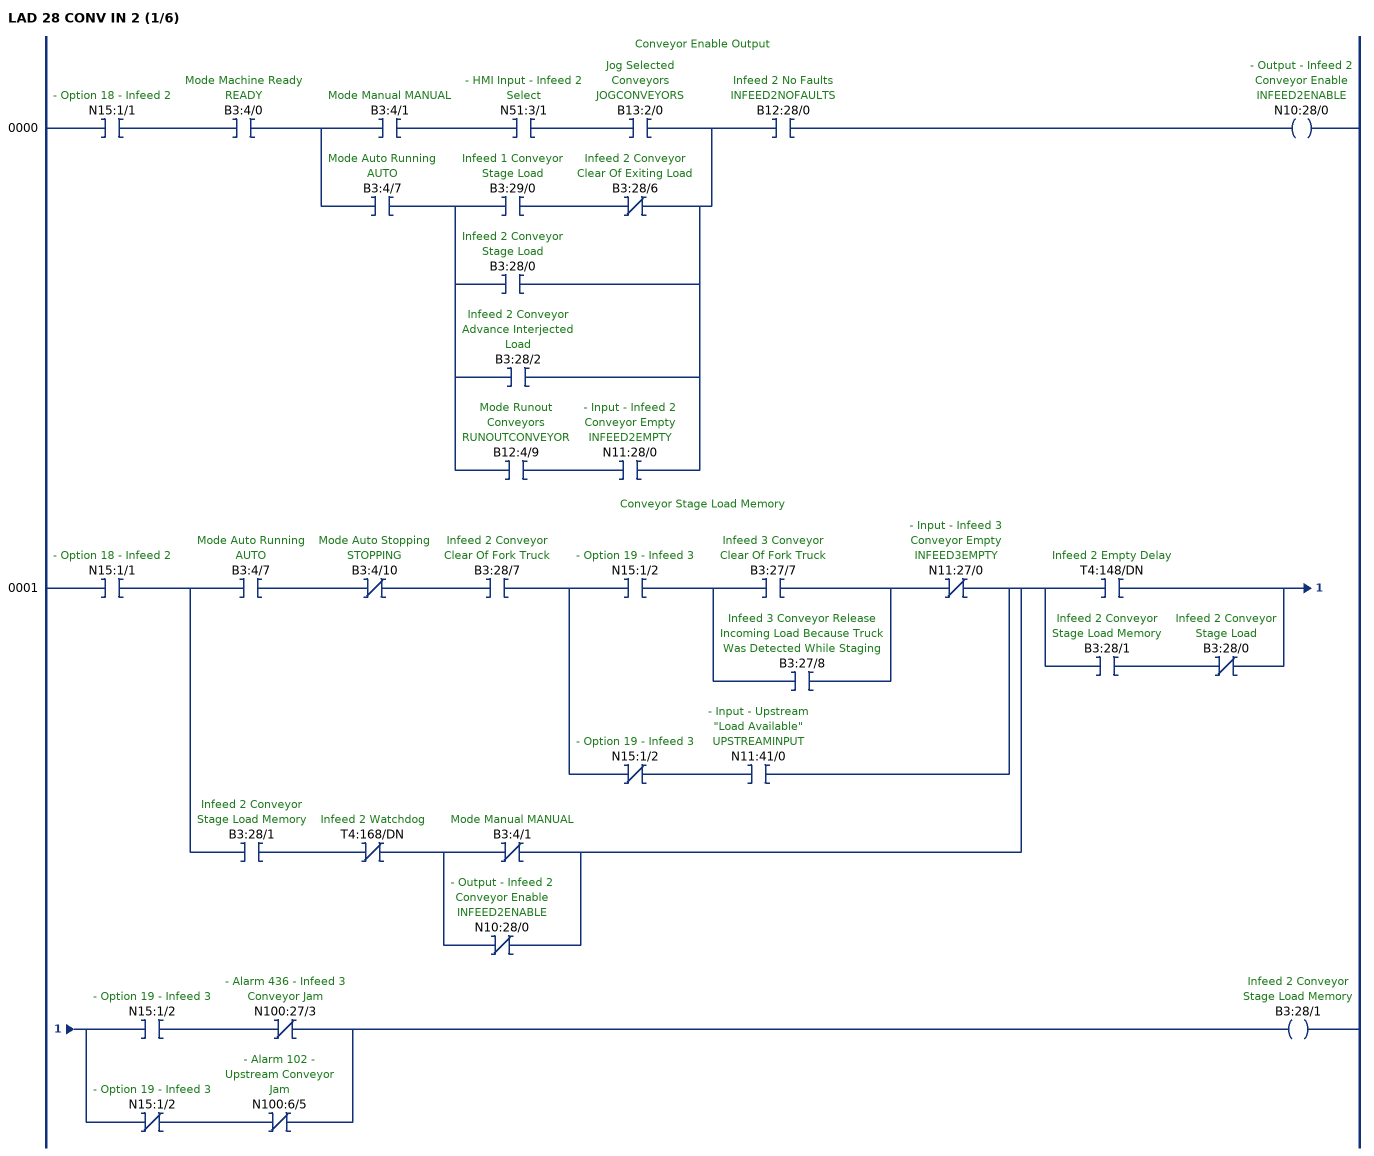
% Rung: 0 %
% Conveyor Enable Output %
SOR XIC N15:1/1 XIC B3:4/0 BST XIC B3:4/1 XIC N51:3/1 XIC B13:2/0 NXB XIC B3:4/7 BST XIC B3:29/0 XIO B3:28/6 NXB XIC B3:28/0 NXB XIC B3:28/2 NXB XIC B12:4/9 XIC N11:28/0 BND BND XIC B12:28/0 OTE N10:28/0 EOR
%   N15:1/1  "- Option 18 - Infeed 2" %
%   B3:4/0  READY  "Mode Machine Ready" %
%   B3:4/1  MANUAL  "Mode Manual" %
%   N51:3/1  "- HMI Input - Infeed 2 Select" %
%   B13:2/0  JOGCONVEYORS  "Jog Selected Conveyors" %
%   B3:4/7  AUTO  "Mode Auto Running" %
%   B3:29/0  "Infeed 1 Conveyor Stage Load" %
%   B3:28/6  "Infeed 2 Conveyor Clear Of Exiting Load" %
%   B3:28/0  "Infeed 2 Conveyor Stage Load" %
%   B3:28/2  "Infeed 2 Conveyor Advance Interjected Load" %
%   B12:4/9  RUNOUTCONVEYOR  "Mode Runout Conveyors" %
%   N11:28/0  INFEED2EMPTY  "- Input - Infeed 2 Conveyor Empty" %
%   B12:28/0  INFEED2NOFAULTS  "Infeed 2 No Faults" %
%   N10:28/0  INFEED2ENABLE  "- Output - Infeed 2 Conveyor Enable" %
% Rung: 1 %
% Conveyor Stage Load Memory %
SOR XIC N15:1/1 BST XIC B3:4/7 XIO B3:4/10 XIC B3:28/7 BST XIC N15:1/2 BST XIC B3:27/7 NXB XIC B3:27/8 BND XIO N11:27/0 NXB XIO N15:1/2 XIC N11:41/0 BND NXB XIC B3:28/1 XIO T4:168/DN BST XIO B3:4/1 NXB XIO N10:28/0 BND BND BST XIC T4:148/DN NXB XIC B3:28/1 XIO B3:28/0 BND BST XIC N15:1/2 XIO N100:27/3 NXB XIO N15:1/2 XIO N100:6/5 BND OTE B3:28/1 EOR
%   N15:1/1  "- Option 18 - Infeed 2" %
%   B3:4/7  AUTO  "Mode Auto Running" %
%   B3:4/10  STOPPING  "Mode Auto Stopping" %
%   B3:28/7  "Infeed 2 Conveyor Clear Of Fork Truck" %
%   N15:1/2  "- Option 19 - Infeed 3" %
%   B3:27/7  "Infeed 3 Conveyor Clear Of Fork Truck" %
%   B3:27/8  "Infeed 3 Conveyor Release Incoming Load Because Truck Was Detected While Staging" %
%   N11:27/0  INFEED3EMPTY  "- Input - Infeed 3 Conveyor Empty" %
%   N11:41/0  UPSTREAMINPUT  "- Input - Upstream "Load Available"" %
%   B3:28/1  "Infeed 2 Conveyor Stage Load Memory" %
%   T4:168  "Infeed 2 Watchdog" %
%   B3:4/1  MANUAL  "Mode Manual" %
%   N10:28/0  INFEED2ENABLE  "- Output - Infeed 2 Conveyor Enable" %
%   T4:148  "Infeed 2 Empty Delay" %
%   B3:28/0  "Infeed 2 Conveyor Stage Load" %
%   N100:27/3  "- Alarm 436 - Infeed 3 Conveyor Jam" %
%   N100:6/5  "- Alarm 102 - Upstream Conveyor Jam" %

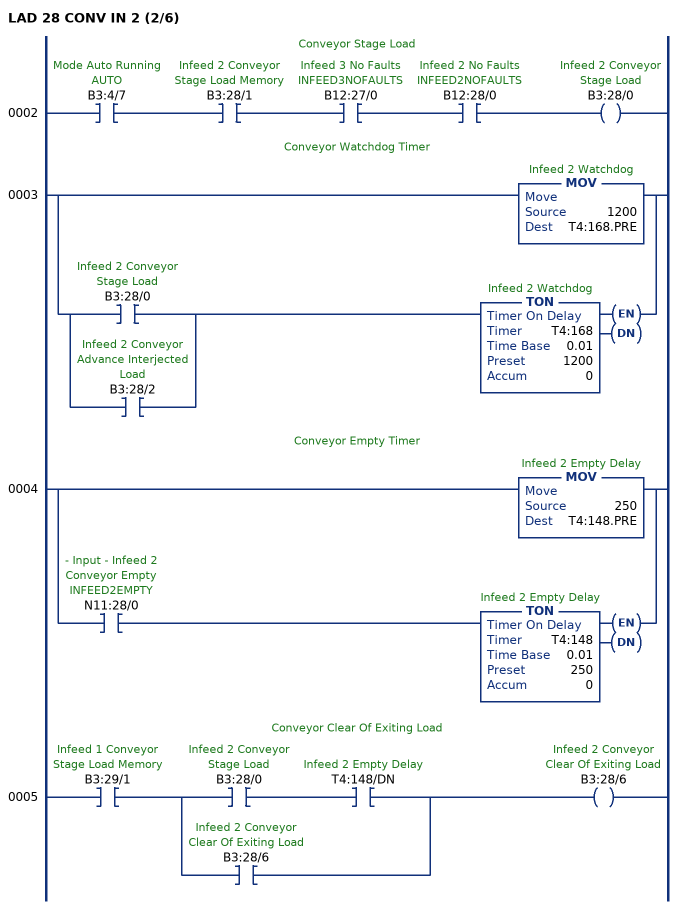
% Rung: 2 %
% Conveyor Stage Load %
SOR XIC B3:4/7 XIC B3:28/1 XIC B12:27/0 XIC B12:28/0 OTE B3:28/0 EOR
%   B3:4/7  AUTO  "Mode Auto Running" %
%   B3:28/1  "Infeed 2 Conveyor Stage Load Memory" %
%   B12:27/0  INFEED3NOFAULTS  "Infeed 3 No Faults" %
%   B12:28/0  INFEED2NOFAULTS  "Infeed 2 No Faults" %
%   B3:28/0  "Infeed 2 Conveyor Stage Load" %
% Rung: 3 %
% Conveyor Watchdog Timer %
SOR BST MOV 1200 T4:168.PRE NXB BST XIC B3:28/0 NXB XIC B3:28/2 BND TON T4:168 0.01 1200 0 BND EOR
%   T4:168  "Infeed 2 Watchdog" %
%   B3:28/0  "Infeed 2 Conveyor Stage Load" %
%   B3:28/2  "Infeed 2 Conveyor Advance Interjected Load" %
% Rung: 4 %
% Conveyor Empty Timer %
SOR BST MOV 250 T4:148.PRE NXB XIC N11:28/0 TON T4:148 0.01 250 0 BND EOR
%   T4:148  "Infeed 2 Empty Delay" %
%   N11:28/0  INFEED2EMPTY  "- Input - Infeed 2 Conveyor Empty" %
% Rung: 5 %
% Conveyor Clear Of Exiting Load %
SOR XIC B3:29/1 BST XIC B3:28/0 XIC T4:148/DN NXB XIC B3:28/6 BND OTE B3:28/6 EOR
%   B3:29/1  "Infeed 1 Conveyor Stage Load Memory" %
%   B3:28/0  "Infeed 2 Conveyor Stage Load" %
%   T4:148  "Infeed 2 Empty Delay" %
%   B3:28/6  "Infeed 2 Conveyor Clear Of Exiting Load" %

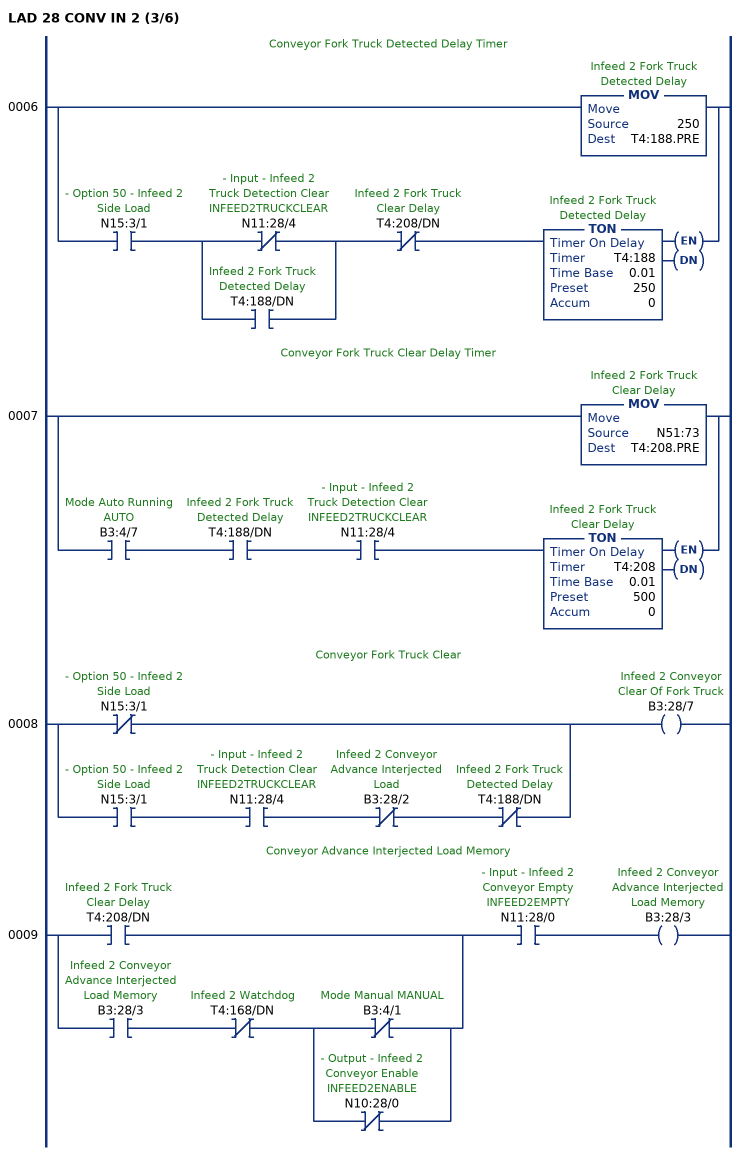
% Rung: 6 %
% Conveyor Fork Truck Detected Delay Timer %
SOR BST MOV 250 T4:188.PRE NXB XIC N15:3/1 BST XIO N11:28/4 NXB XIC T4:188/DN BND XIO T4:208/DN TON T4:188 0.01 250 0 BND EOR
%   T4:188  "Infeed 2 Fork Truck Detected Delay" %
%   N15:3/1  "- Option 50 - Infeed 2 Side Load" %
%   N11:28/4  INFEED2TRUCKCLEAR  "- Input - Infeed 2 Truck Detection Clear" %
%   T4:208  "Infeed 2 Fork Truck Clear Delay" %
% Rung: 7 %
% Conveyor Fork Truck Clear Delay Timer %
SOR BST MOV N51:73 T4:208.PRE NXB XIC B3:4/7 XIC T4:188/DN XIC N11:28/4 TON T4:208 0.01 500 0 BND EOR
%   N51:73  "- HMI Input - Preset Truck Clear" %
%   T4:208  "Infeed 2 Fork Truck Clear Delay" %
%   B3:4/7  AUTO  "Mode Auto Running" %
%   T4:188  "Infeed 2 Fork Truck Detected Delay" %
%   N11:28/4  INFEED2TRUCKCLEAR  "- Input - Infeed 2 Truck Detection Clear" %
% Rung: 8 %
% Conveyor Fork Truck Clear %
SOR BST XIO N15:3/1 NXB XIC N15:3/1 XIC N11:28/4 XIO B3:28/2 XIO T4:188/DN BND OTE B3:28/7 EOR
%   N15:3/1  "- Option 50 - Infeed 2 Side Load" %
%   N11:28/4  INFEED2TRUCKCLEAR  "- Input - Infeed 2 Truck Detection Clear" %
%   B3:28/2  "Infeed 2 Conveyor Advance Interjected Load" %
%   T4:188  "Infeed 2 Fork Truck Detected Delay" %
%   B3:28/7  "Infeed 2 Conveyor Clear Of Fork Truck" %
% Rung: 9 %
% Conveyor Advance Interjected Load Memory %
SOR BST XIC T4:208/DN NXB XIC B3:28/3 XIO T4:168/DN BST XIO B3:4/1 NXB XIO N10:28/0 BND BND XIC N11:28/0 OTE B3:28/3 EOR
%   T4:208  "Infeed 2 Fork Truck Clear Delay" %
%   B3:28/3  "Infeed 2 Conveyor Advance Interjected Load Memory" %
%   T4:168  "Infeed 2 Watchdog" %
%   B3:4/1  MANUAL  "Mode Manual" %
%   N10:28/0  INFEED2ENABLE  "- Output - Infeed 2 Conveyor Enable" %
%   N11:28/0  INFEED2EMPTY  "- Input - Infeed 2 Conveyor Empty" %

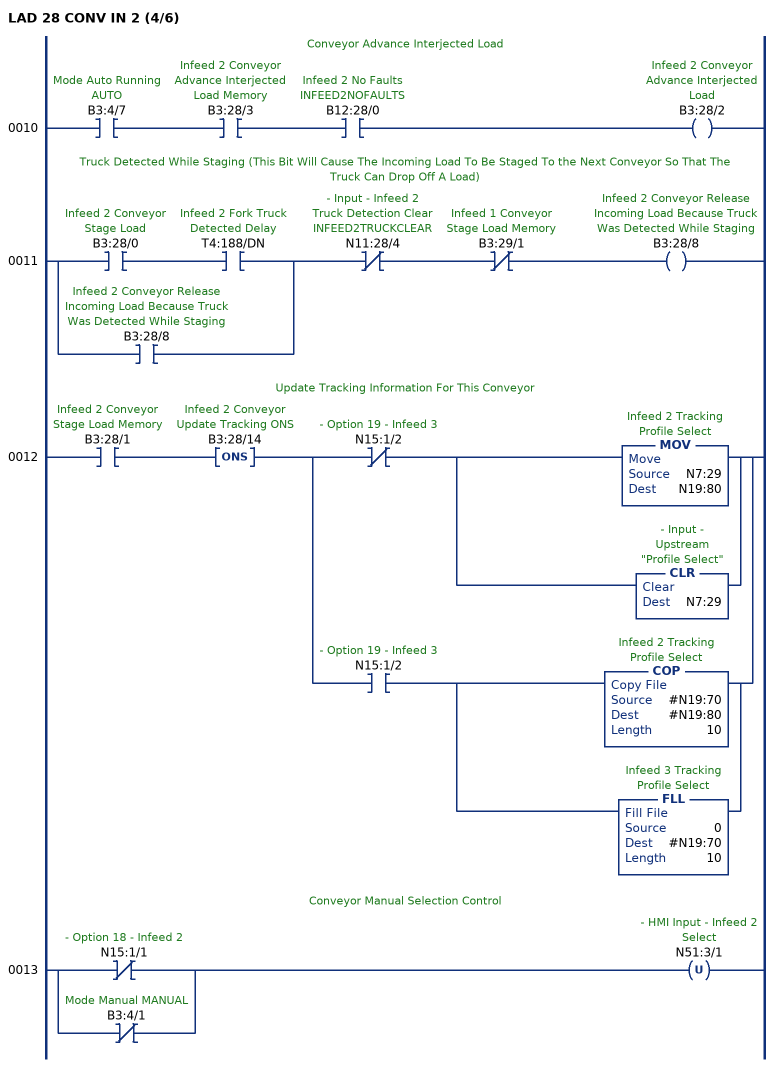
% Rung: 10 %
% Conveyor Advance Interjected Load %
SOR XIC B3:4/7 XIC B3:28/3 XIC B12:28/0 OTE B3:28/2 EOR
%   B3:4/7  AUTO  "Mode Auto Running" %
%   B3:28/3  "Infeed 2 Conveyor Advance Interjected Load Memory" %
%   B12:28/0  INFEED2NOFAULTS  "Infeed 2 No Faults" %
%   B3:28/2  "Infeed 2 Conveyor Advance Interjected Load" %
% Rung: 11 %
% Truck Detected While Staging (This Bit Will Cause The Incoming Load To Be Staged To the Next Conveyor So That The Truck Can Drop Off A Load) %
SOR BST XIC B3:28/0 XIC T4:188/DN NXB XIC B3:28/8 BND XIO N11:28/4 XIO B3:29/1 OTE B3:28/8 EOR
%   B3:28/0  "Infeed 2 Conveyor Stage Load" %
%   T4:188  "Infeed 2 Fork Truck Detected Delay" %
%   B3:28/8  "Infeed 2 Conveyor Release Incoming Load Because Truck Was Detected While Staging" %
%   N11:28/4  INFEED2TRUCKCLEAR  "- Input - Infeed 2 Truck Detection Clear" %
%   B3:29/1  "Infeed 1 Conveyor Stage Load Memory" %
% Rung: 12 %
% Update Tracking Information For This Conveyor %
SOR XIC B3:28/1 ONS B3:28/14 BST XIO N15:1/2 BST MOV N7:29 N19:80 NXB CLR N7:29 BND NXB XIC N15:1/2 BST COP #N19:70 #N19:80 10 NXB FLL 0 #N19:70 10 BND BND EOR
%   B3:28/1  "Infeed 2 Conveyor Stage Load Memory" %
%   B3:28/14  "Infeed 2 Conveyor Update Tracking ONS" %
%   N15:1/2  "- Option 19 - Infeed 3" %
%   N7:29  "- Input - Upstream "Profile Select"" %
%   N19:80  "Infeed 2 Tracking Profile Select" %
%   N19:70  "Infeed 3 Tracking Profile Select" %
% Rung: 13 %
% Conveyor Manual Selection Control %
SOR BST XIO N15:1/1 NXB XIO B3:4/1 BND OTU N51:3/1 EOR
%   N15:1/1  "- Option 18 - Infeed 2" %
%   B3:4/1  MANUAL  "Mode Manual" %
%   N51:3/1  "- HMI Input - Infeed 2 Select" %

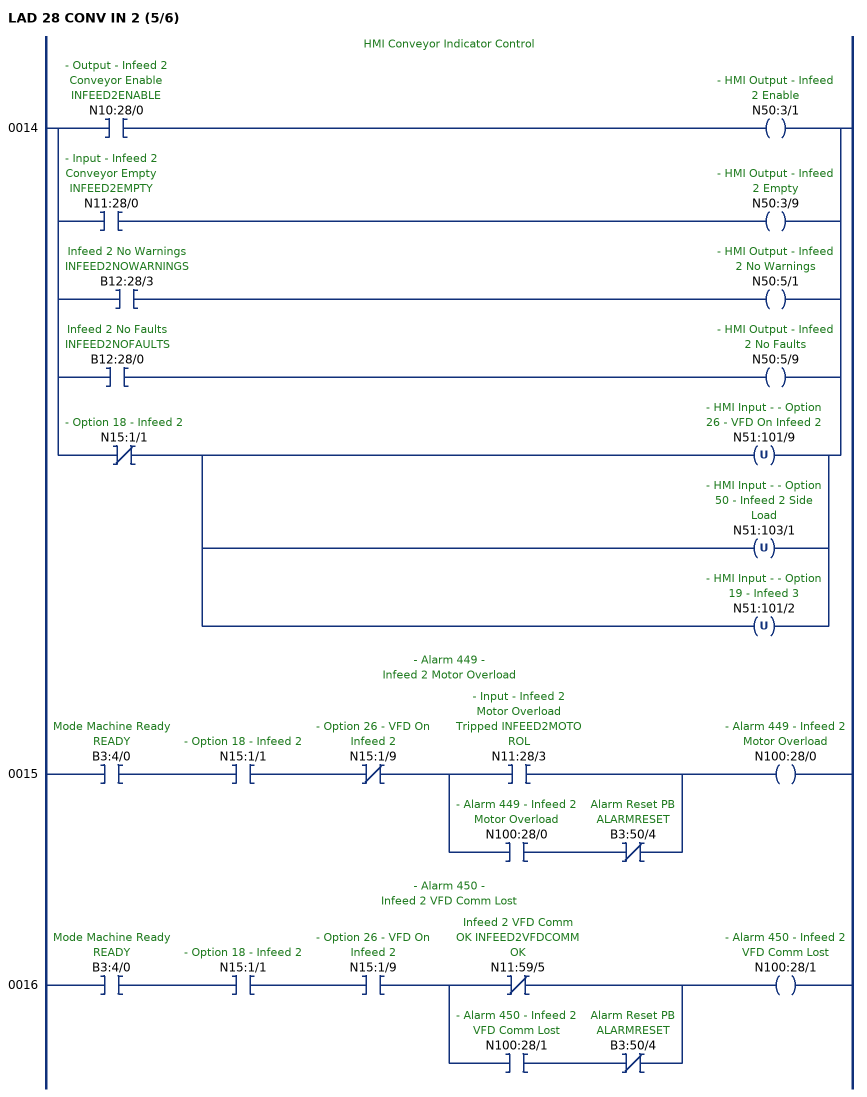
% Rung: 14 %
% HMI Conveyor Indicator Control %
SOR BST XIC N10:28/0 OTE N50:3/1 NXB XIC N11:28/0 OTE N50:3/9 NXB XIC B12:28/3 OTE N50:5/1 NXB XIC B12:28/0 OTE N50:5/9 NXB XIO N15:1/1 BST OTU N51:101/9 NXB OTU N51:103/1 NXB OTU N51:101/2 BND BND EOR
%   N10:28/0  INFEED2ENABLE  "- Output - Infeed 2 Conveyor Enable" %
%   N50:3/1  "- HMI Output - Infeed 2 Enable" %
%   N11:28/0  INFEED2EMPTY  "- Input - Infeed 2 Conveyor Empty" %
%   N50:3/9  "- HMI Output - Infeed 2 Empty" %
%   B12:28/3  INFEED2NOWARNINGS  "Infeed 2 No Warnings" %
%   N50:5/1  "- HMI Output - Infeed 2 No Warnings" %
%   B12:28/0  INFEED2NOFAULTS  "Infeed 2 No Faults" %
%   N50:5/9  "- HMI Output - Infeed 2 No Faults" %
%   N15:1/1  "- Option 18 - Infeed 2" %
%   N51:101/9  "- HMI Input - - Option 26 - VFD On Infeed 2" %
%   N51:103/1  "- HMI Input - - Option 50 - Infeed 2 Side Load" %
%   N51:101/2  "- HMI Input - - Option 19 - Infeed 3" %
% Rung: 15 %
% - Alarm 449 -
% 
% Infeed 2 Motor Overload %
SOR XIC B3:4/0 XIC N15:1/1 XIO N15:1/9 BST XIC N11:28/3 NXB XIC N100:28/0 XIO B3:50/4 BND OTE N100:28/0 EOR
%   B3:4/0  READY  "Mode Machine Ready" %
%   N15:1/1  "- Option 18 - Infeed 2" %
%   N15:1/9  "- Option 26 - VFD On Infeed 2" %
%   N11:28/3  INFEED2MOTOROL  "- Input - Infeed 2 Motor Overload Tripped" %
%   N100:28/0  "- Alarm 449 - Infeed 2 Motor Overload" %
%   B3:50/4  ALARMRESET  "Alarm Reset PB" %
% Rung: 16 %
% - Alarm 450 -
% 
% Infeed 2 VFD Comm Lost %
SOR XIC B3:4/0 XIC N15:1/1 XIC N15:1/9 BST XIO N11:59/5 NXB XIC N100:28/1 XIO B3:50/4 BND OTE N100:28/1 EOR
%   B3:4/0  READY  "Mode Machine Ready" %
%   N15:1/1  "- Option 18 - Infeed 2" %
%   N15:1/9  "- Option 26 - VFD On Infeed 2" %
%   N11:59/5  INFEED2VFDCOMMOK  "Infeed 2 VFD Comm OK" %
%   N100:28/1  "- Alarm 450 - Infeed 2 VFD Comm Lost" %
%   B3:50/4  ALARMRESET  "Alarm Reset PB" %

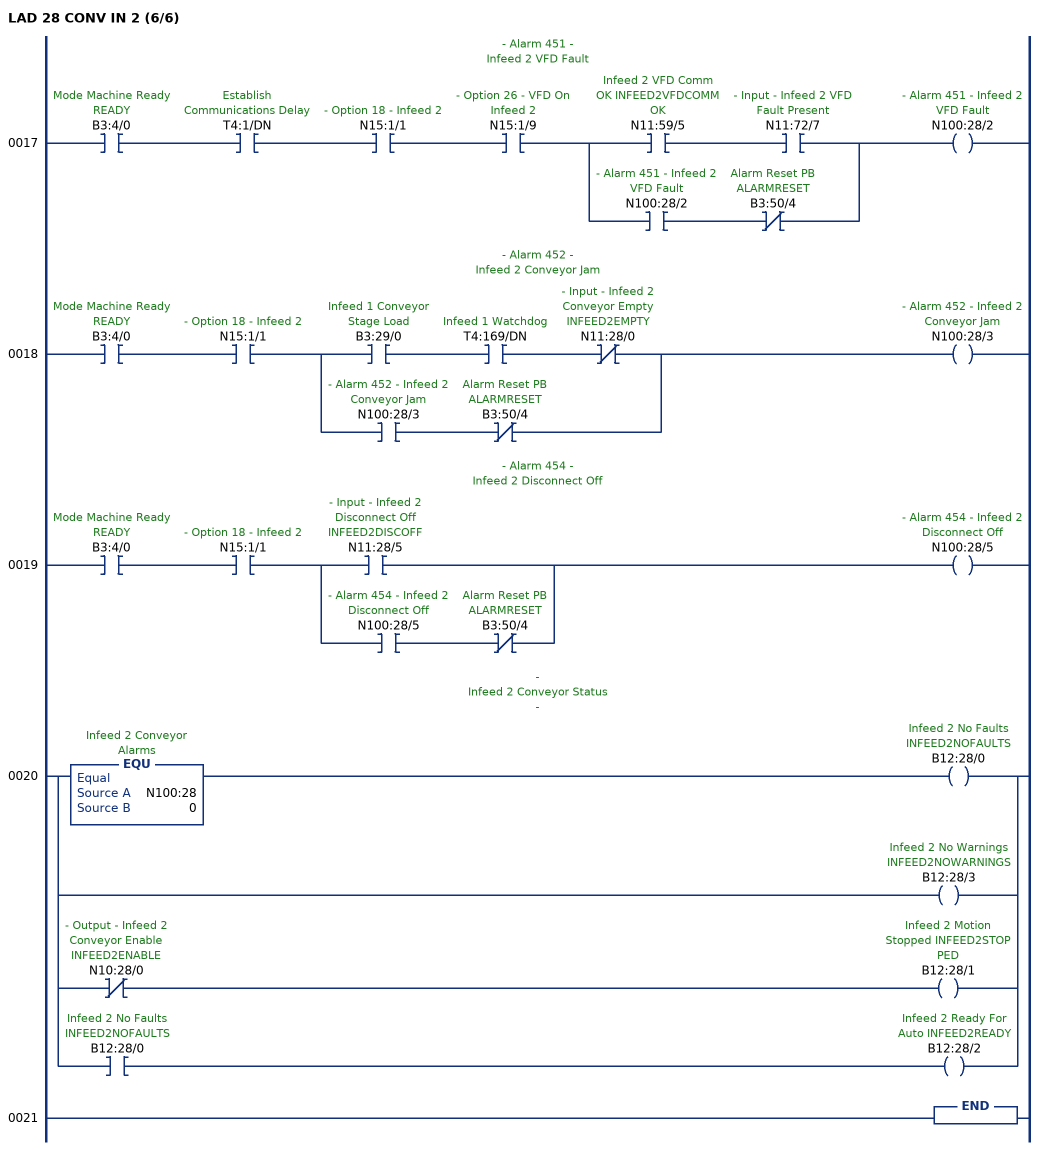
% Rung: 17 %
% - Alarm 451 -
% 
% Infeed 2 VFD Fault %
SOR XIC B3:4/0 XIC T4:1/DN XIC N15:1/1 XIC N15:1/9 BST XIC N11:59/5 XIC N11:72/7 NXB XIC N100:28/2 XIO B3:50/4 BND OTE N100:28/2 EOR
%   B3:4/0  READY  "Mode Machine Ready" %
%   T4:1  "Establish Communications Delay" %
%   N15:1/1  "- Option 18 - Infeed 2" %
%   N15:1/9  "- Option 26 - VFD On Infeed 2" %
%   N11:59/5  INFEED2VFDCOMMOK  "Infeed 2 VFD Comm OK" %
%   N11:72/7  "- Input - Infeed 2 VFD Fault Present" %
%   N100:28/2  "- Alarm 451 - Infeed 2 VFD Fault" %
%   B3:50/4  ALARMRESET  "Alarm Reset PB" %
% Rung: 18 %
% - Alarm 452 -
% 
% Infeed 2 Conveyor Jam %
SOR XIC B3:4/0 XIC N15:1/1 BST XIC B3:29/0 XIC T4:169/DN XIO N11:28/0 NXB XIC N100:28/3 XIO B3:50/4 BND OTE N100:28/3 EOR
%   B3:4/0  READY  "Mode Machine Ready" %
%   N15:1/1  "- Option 18 - Infeed 2" %
%   B3:29/0  "Infeed 1 Conveyor Stage Load" %
%   T4:169  "Infeed 1 Watchdog" %
%   N11:28/0  INFEED2EMPTY  "- Input - Infeed 2 Conveyor Empty" %
%   N100:28/3  "- Alarm 452 - Infeed 2 Conveyor Jam" %
%   B3:50/4  ALARMRESET  "Alarm Reset PB" %
% Rung: 19 %
% - Alarm 454 -
% 
% Infeed 2 Disconnect Off %
SOR XIC B3:4/0 XIC N15:1/1 BST XIC N11:28/5 NXB XIC N100:28/5 XIO B3:50/4 BND OTE N100:28/5 EOR
%   B3:4/0  READY  "Mode Machine Ready" %
%   N15:1/1  "- Option 18 - Infeed 2" %
%   N11:28/5  INFEED2DISCOFF  "- Input - Infeed 2 Disconnect Off" %
%   N100:28/5  "- Alarm 454 - Infeed 2 Disconnect Off" %
%   B3:50/4  ALARMRESET  "Alarm Reset PB" %
% Rung: 20 %
% -
% 
% Infeed 2 Conveyor Status
% 
% - %
SOR BST EQU N100:28 0 OTE B12:28/0 NXB OTE B12:28/3 NXB XIO N10:28/0 OTE B12:28/1 NXB XIC B12:28/0 OTE B12:28/2 BND EOR
%   N100:28  "Infeed 2 Conveyor Alarms" %
%   B12:28/0  INFEED2NOFAULTS  "Infeed 2 No Faults" %
%   B12:28/3  INFEED2NOWARNINGS  "Infeed 2 No Warnings" %
%   N10:28/0  INFEED2ENABLE  "- Output - Infeed 2 Conveyor Enable" %
%   B12:28/1  INFEED2STOPPED  "Infeed 2 Motion Stopped" %
%   B12:28/2  INFEED2READY  "Infeed 2 Ready For Auto" %
% Rung: 21 %
SOR END EOR

LADDER 29 "CONV IN 1"
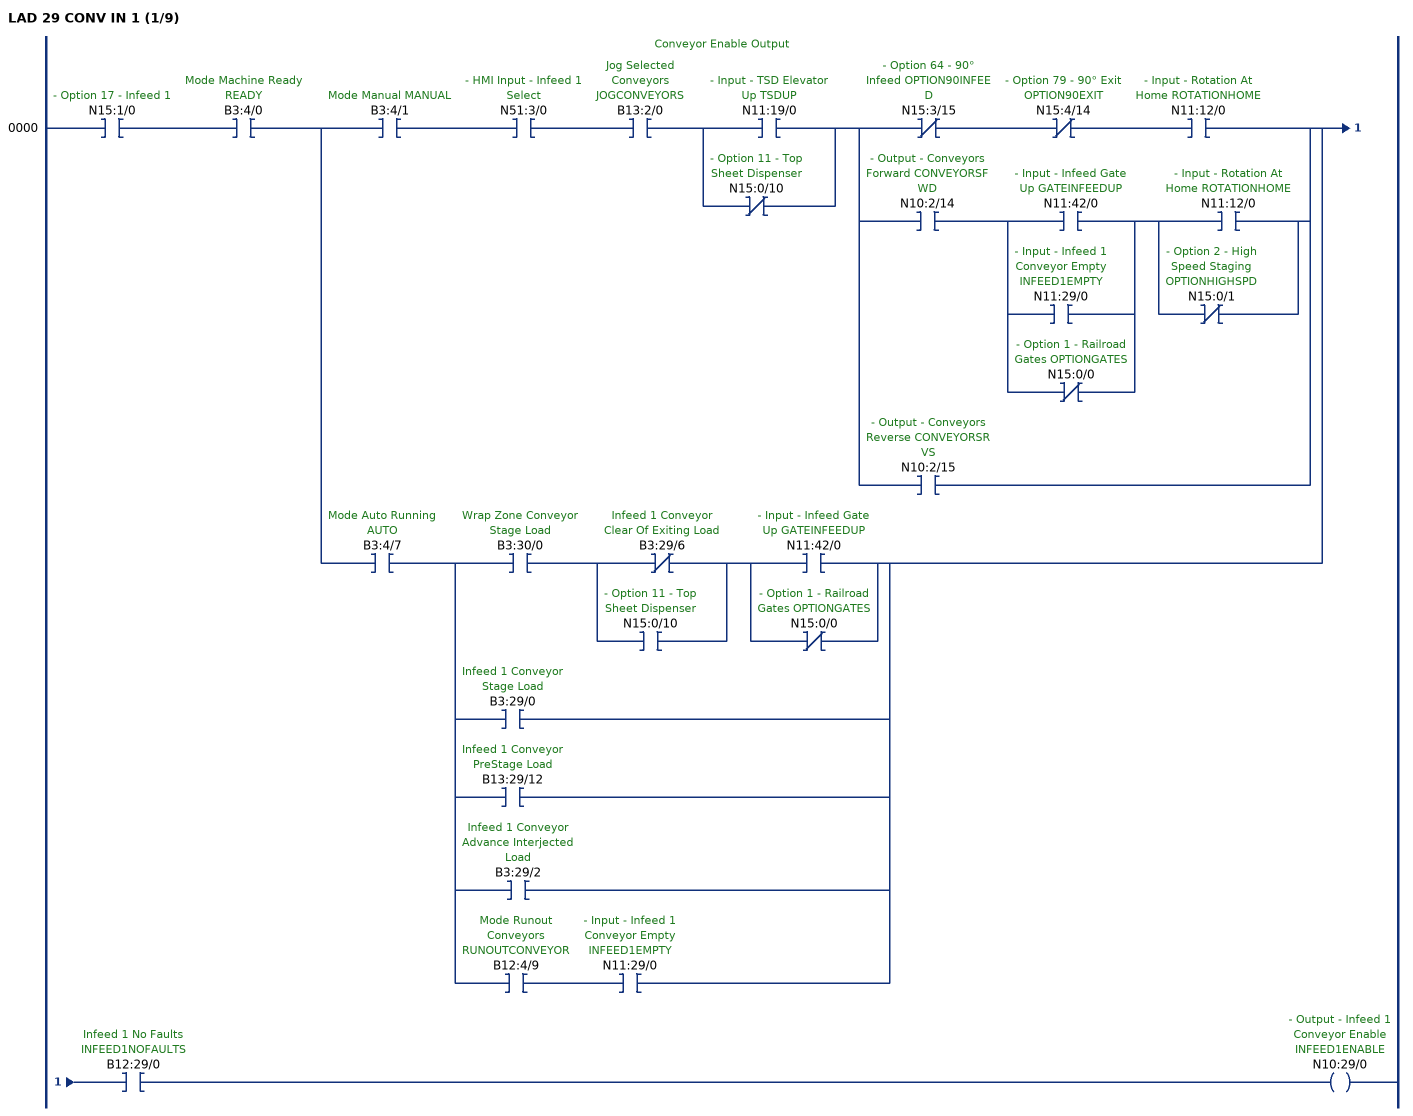
% Rung: 0 %
% Conveyor Enable Output %
SOR XIC N15:1/0 XIC B3:4/0 BST XIC B3:4/1 XIC N51:3/0 XIC B13:2/0 BST XIC N11:19/0 NXB XIO N15:0/10 BND BST XIO N15:3/15 XIO N15:4/14 XIC N11:12/0 NXB XIC N10:2/14 BST XIC N11:42/0 NXB XIC N11:29/0 NXB XIO N15:0/0 BND BST XIC N11:12/0 NXB XIO N15:0/1 BND NXB XIC N10:2/15 BND NXB XIC B3:4/7 BST XIC B3:30/0 BST XIO B3:29/6 NXB XIC N15:0/10 BND BST XIC N11:42/0 NXB XIO N15:0/0 BND NXB XIC B3:29/0 NXB XIC B13:29/12 NXB XIC B3:29/2 NXB XIC B12:4/9 XIC N11:29/0 BND BND XIC B12:29/0 OTE N10:29/0 EOR
%   N15:1/0  "- Option 17 - Infeed 1" %
%   B3:4/0  READY  "Mode Machine Ready" %
%   B3:4/1  MANUAL  "Mode Manual" %
%   N51:3/0  "- HMI Input - Infeed 1 Select" %
%   B13:2/0  JOGCONVEYORS  "Jog Selected Conveyors" %
%   N11:19/0  TSDUP  "- Input - TSD Elevator Up" %
%   N15:0/10  "- Option 11 - Top Sheet Dispenser" %
%   N15:3/15  OPTION90INFEED  "- Option 64 - 90° Infeed" %
%   N15:4/14  OPTION90EXIT  "- Option 79 - 90° Exit" %
%   N11:12/0  ROTATIONHOME  "- Input - Rotation At Home" %
%   N10:2/14  CONVEYORSFWD  "- Output - Conveyors Forward" %
%   N11:42/0  GATEINFEEDUP  "- Input - Infeed Gate Up" %
%   N11:29/0  INFEED1EMPTY  "- Input - Infeed 1 Conveyor Empty" %
%   N15:0/0  OPTIONGATES  "- Option 1 - Railroad Gates" %
%   N15:0/1  OPTIONHIGHSPD  "- Option 2 - High Speed Staging" %
%   N10:2/15  CONVEYORSRVS  "- Output - Conveyors Reverse" %
%   B3:4/7  AUTO  "Mode Auto Running" %
%   B3:30/0  "Wrap Zone Conveyor Stage Load" %
%   B3:29/6  "Infeed 1 Conveyor Clear Of Exiting Load" %
%   B3:29/0  "Infeed 1 Conveyor Stage Load" %
%   B13:29/12  "Infeed 1 Conveyor PreStage Load" %
%   B3:29/2  "Infeed 1 Conveyor Advance Interjected Load" %
%   B12:4/9  RUNOUTCONVEYOR  "Mode Runout Conveyors" %
%   B12:29/0  INFEED1NOFAULTS  "Infeed 1 No Faults" %
%   N10:29/0  INFEED1ENABLE  "- Output - Infeed 1 Conveyor Enable" %

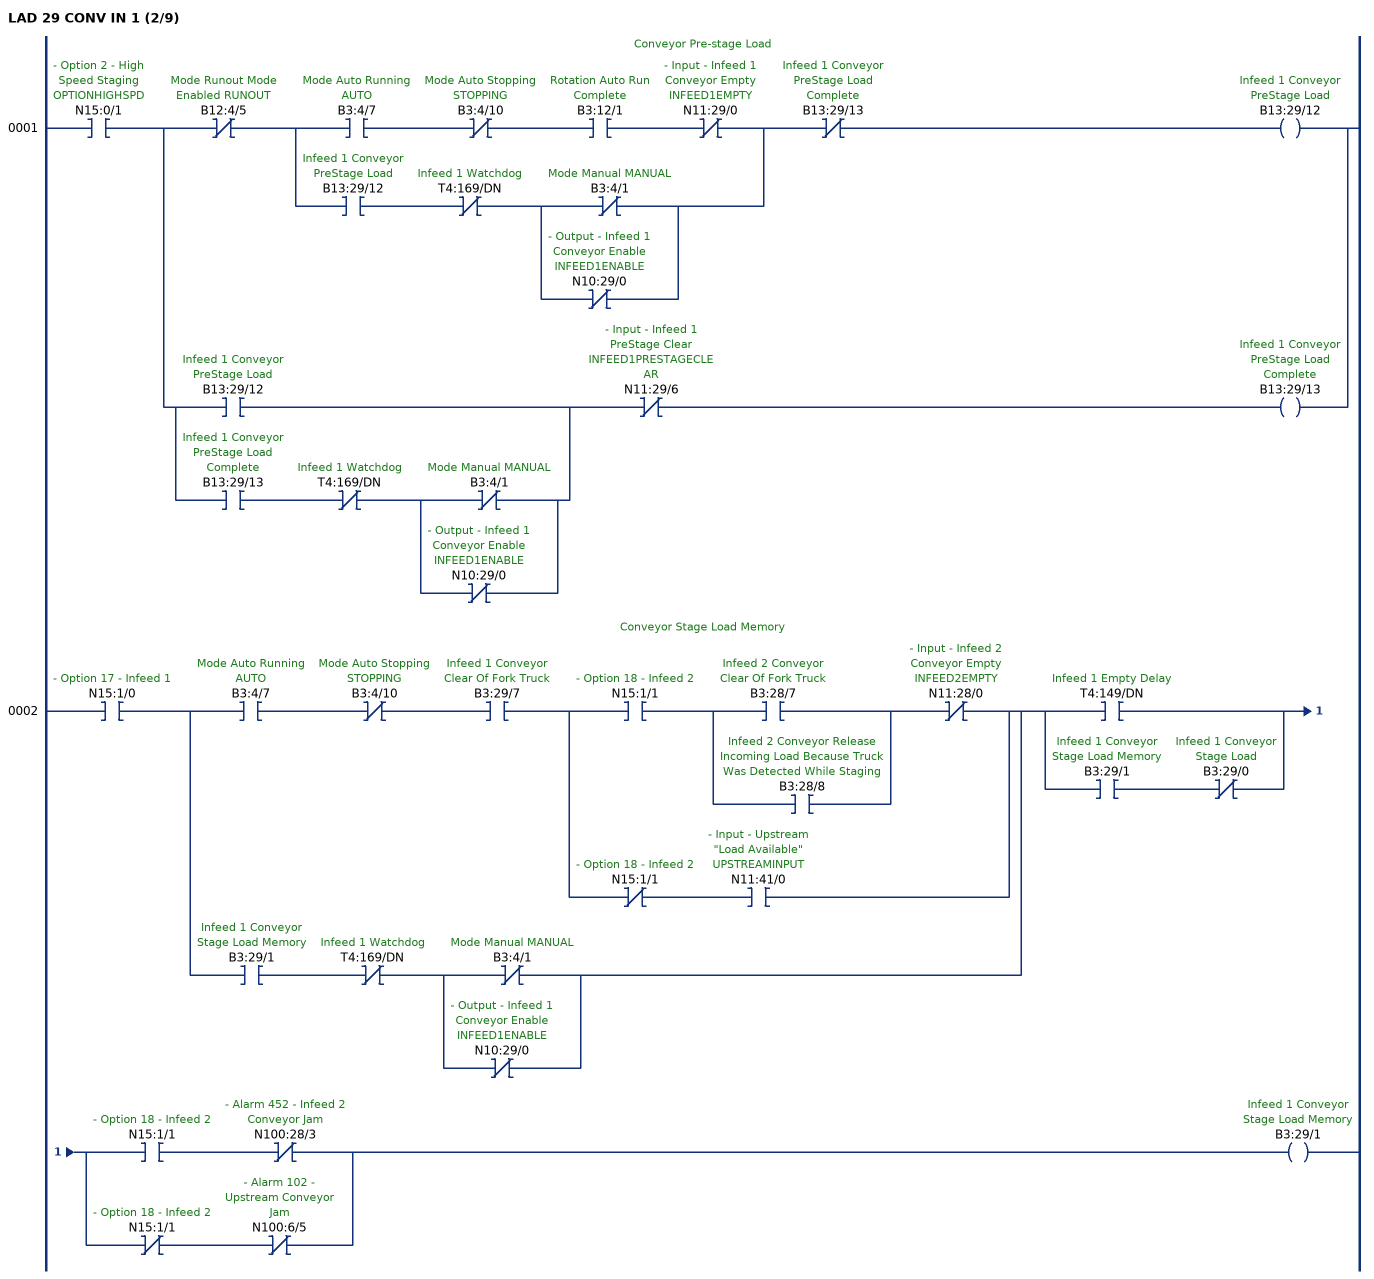
% Rung: 1 %
% Conveyor Pre-stage Load %
SOR XIC N15:0/1 BST XIO B12:4/5 BST XIC B3:4/7 XIO B3:4/10 XIC B3:12/1 XIO N11:29/0 NXB XIC B13:29/12 XIO T4:169/DN BST XIO B3:4/1 NXB XIO N10:29/0 BND BND XIO B13:29/13 OTE B13:29/12 NXB BST XIC B13:29/12 NXB XIC B13:29/13 XIO T4:169/DN BST XIO B3:4/1 NXB XIO N10:29/0 BND BND XIO N11:29/6 OTE B13:29/13 BND EOR
%   N15:0/1  OPTIONHIGHSPD  "- Option 2 - High Speed Staging" %
%   B12:4/5  RUNOUT  "Mode Runout Mode Enabled" %
%   B3:4/7  AUTO  "Mode Auto Running" %
%   B3:4/10  STOPPING  "Mode Auto Stopping" %
%   B3:12/1  "Rotation Auto Run Complete" %
%   N11:29/0  INFEED1EMPTY  "- Input - Infeed 1 Conveyor Empty" %
%   B13:29/12  "Infeed 1 Conveyor PreStage Load" %
%   T4:169  "Infeed 1 Watchdog" %
%   B3:4/1  MANUAL  "Mode Manual" %
%   N10:29/0  INFEED1ENABLE  "- Output - Infeed 1 Conveyor Enable" %
%   B13:29/13  "Infeed 1 Conveyor PreStage Load Complete" %
%   N11:29/6  INFEED1PRESTAGECLEAR  "- Input - Infeed 1 PreStage Clear" %
% Rung: 2 %
% Conveyor Stage Load Memory %
SOR XIC N15:1/0 BST XIC B3:4/7 XIO B3:4/10 XIC B3:29/7 BST XIC N15:1/1 BST XIC B3:28/7 NXB XIC B3:28/8 BND XIO N11:28/0 NXB XIO N15:1/1 XIC N11:41/0 BND NXB XIC B3:29/1 XIO T4:169/DN BST XIO B3:4/1 NXB XIO N10:29/0 BND BND BST XIC T4:149/DN NXB XIC B3:29/1 XIO B3:29/0 BND BST XIC N15:1/1 XIO N100:28/3 NXB XIO N15:1/1 XIO N100:6/5 BND OTE B3:29/1 EOR
%   N15:1/0  "- Option 17 - Infeed 1" %
%   B3:4/7  AUTO  "Mode Auto Running" %
%   B3:4/10  STOPPING  "Mode Auto Stopping" %
%   B3:29/7  "Infeed 1 Conveyor Clear Of Fork Truck" %
%   N15:1/1  "- Option 18 - Infeed 2" %
%   B3:28/7  "Infeed 2 Conveyor Clear Of Fork Truck" %
%   B3:28/8  "Infeed 2 Conveyor Release Incoming Load Because Truck Was Detected While Staging" %
%   N11:28/0  INFEED2EMPTY  "- Input - Infeed 2 Conveyor Empty" %
%   N11:41/0  UPSTREAMINPUT  "- Input - Upstream "Load Available"" %
%   B3:29/1  "Infeed 1 Conveyor Stage Load Memory" %
%   T4:169  "Infeed 1 Watchdog" %
%   B3:4/1  MANUAL  "Mode Manual" %
%   N10:29/0  INFEED1ENABLE  "- Output - Infeed 1 Conveyor Enable" %
%   T4:149  "Infeed 1 Empty Delay" %
%   B3:29/0  "Infeed 1 Conveyor Stage Load" %
%   N100:28/3  "- Alarm 452 - Infeed 2 Conveyor Jam" %
%   N100:6/5  "- Alarm 102 - Upstream Conveyor Jam" %

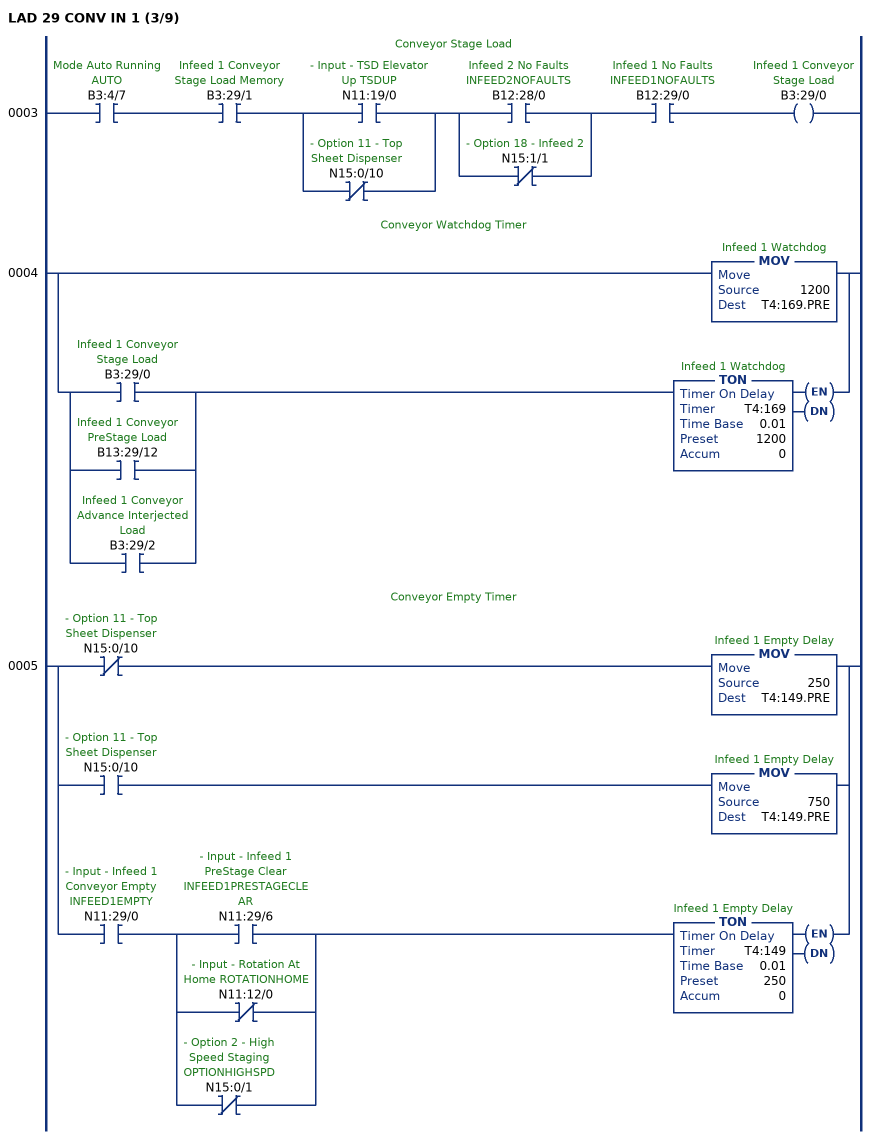
% Rung: 3 %
% Conveyor Stage Load %
SOR XIC B3:4/7 XIC B3:29/1 BST XIC N11:19/0 NXB XIO N15:0/10 BND BST XIC B12:28/0 NXB XIO N15:1/1 BND XIC B12:29/0 OTE B3:29/0 EOR
%   B3:4/7  AUTO  "Mode Auto Running" %
%   B3:29/1  "Infeed 1 Conveyor Stage Load Memory" %
%   N11:19/0  TSDUP  "- Input - TSD Elevator Up" %
%   N15:0/10  "- Option 11 - Top Sheet Dispenser" %
%   B12:28/0  INFEED2NOFAULTS  "Infeed 2 No Faults" %
%   N15:1/1  "- Option 18 - Infeed 2" %
%   B12:29/0  INFEED1NOFAULTS  "Infeed 1 No Faults" %
%   B3:29/0  "Infeed 1 Conveyor Stage Load" %
% Rung: 4 %
% Conveyor Watchdog Timer %
SOR BST MOV 1200 T4:169.PRE NXB BST XIC B3:29/0 NXB XIC B13:29/12 NXB XIC B3:29/2 BND TON T4:169 0.01 1200 0 BND EOR
%   T4:169  "Infeed 1 Watchdog" %
%   B3:29/0  "Infeed 1 Conveyor Stage Load" %
%   B13:29/12  "Infeed 1 Conveyor PreStage Load" %
%   B3:29/2  "Infeed 1 Conveyor Advance Interjected Load" %
% Rung: 5 %
% Conveyor Empty Timer %
SOR BST BST XIO N15:0/10 MOV 250 T4:149.PRE NXB XIC N15:0/10 MOV 750 T4:149.PRE BND NXB XIC N11:29/0 BST XIC N11:29/6 NXB XIO N11:12/0 NXB XIO N15:0/1 BND TON T4:149 0.01 250 0 BND EOR
%   N15:0/10  "- Option 11 - Top Sheet Dispenser" %
%   T4:149  "Infeed 1 Empty Delay" %
%   N11:29/0  INFEED1EMPTY  "- Input - Infeed 1 Conveyor Empty" %
%   N11:29/6  INFEED1PRESTAGECLEAR  "- Input - Infeed 1 PreStage Clear" %
%   N11:12/0  ROTATIONHOME  "- Input - Rotation At Home" %
%   N15:0/1  OPTIONHIGHSPD  "- Option 2 - High Speed Staging" %

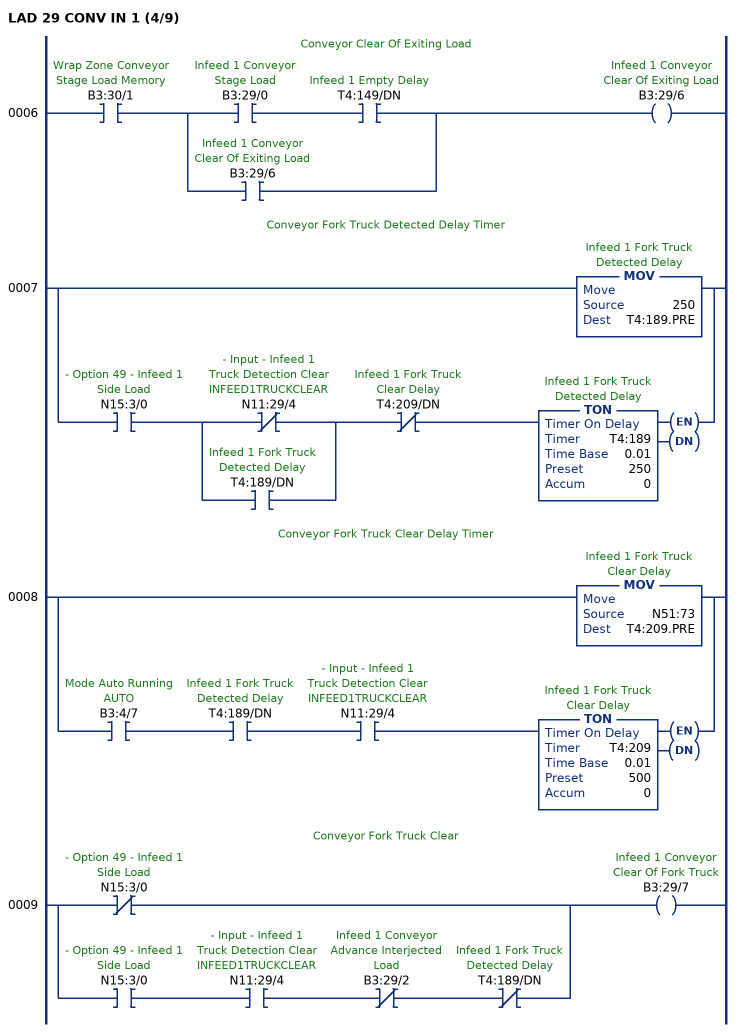
% Rung: 6 %
% Conveyor Clear Of Exiting Load %
SOR XIC B3:30/1 BST XIC B3:29/0 XIC T4:149/DN NXB XIC B3:29/6 BND OTE B3:29/6 EOR
%   B3:30/1  "Wrap Zone Conveyor Stage Load Memory" %
%   B3:29/0  "Infeed 1 Conveyor Stage Load" %
%   T4:149  "Infeed 1 Empty Delay" %
%   B3:29/6  "Infeed 1 Conveyor Clear Of Exiting Load" %
% Rung: 7 %
% Conveyor Fork Truck Detected Delay Timer %
SOR BST MOV 250 T4:189.PRE NXB XIC N15:3/0 BST XIO N11:29/4 NXB XIC T4:189/DN BND XIO T4:209/DN TON T4:189 0.01 250 0 BND EOR
%   T4:189  "Infeed 1 Fork Truck Detected Delay" %
%   N15:3/0  "- Option 49 - Infeed 1 Side Load" %
%   N11:29/4  INFEED1TRUCKCLEAR  "- Input - Infeed 1 Truck Detection Clear" %
%   T4:209  "Infeed 1 Fork Truck Clear Delay" %
% Rung: 8 %
% Conveyor Fork Truck Clear Delay Timer %
SOR BST MOV N51:73 T4:209.PRE NXB XIC B3:4/7 XIC T4:189/DN XIC N11:29/4 TON T4:209 0.01 500 0 BND EOR
%   N51:73  "- HMI Input - Preset Truck Clear" %
%   T4:209  "Infeed 1 Fork Truck Clear Delay" %
%   B3:4/7  AUTO  "Mode Auto Running" %
%   T4:189  "Infeed 1 Fork Truck Detected Delay" %
%   N11:29/4  INFEED1TRUCKCLEAR  "- Input - Infeed 1 Truck Detection Clear" %
% Rung: 9 %
% Conveyor Fork Truck Clear %
SOR BST XIO N15:3/0 NXB XIC N15:3/0 XIC N11:29/4 XIO B3:29/2 XIO T4:189/DN BND OTE B3:29/7 EOR
%   N15:3/0  "- Option 49 - Infeed 1 Side Load" %
%   N11:29/4  INFEED1TRUCKCLEAR  "- Input - Infeed 1 Truck Detection Clear" %
%   B3:29/2  "Infeed 1 Conveyor Advance Interjected Load" %
%   T4:189  "Infeed 1 Fork Truck Detected Delay" %
%   B3:29/7  "Infeed 1 Conveyor Clear Of Fork Truck" %

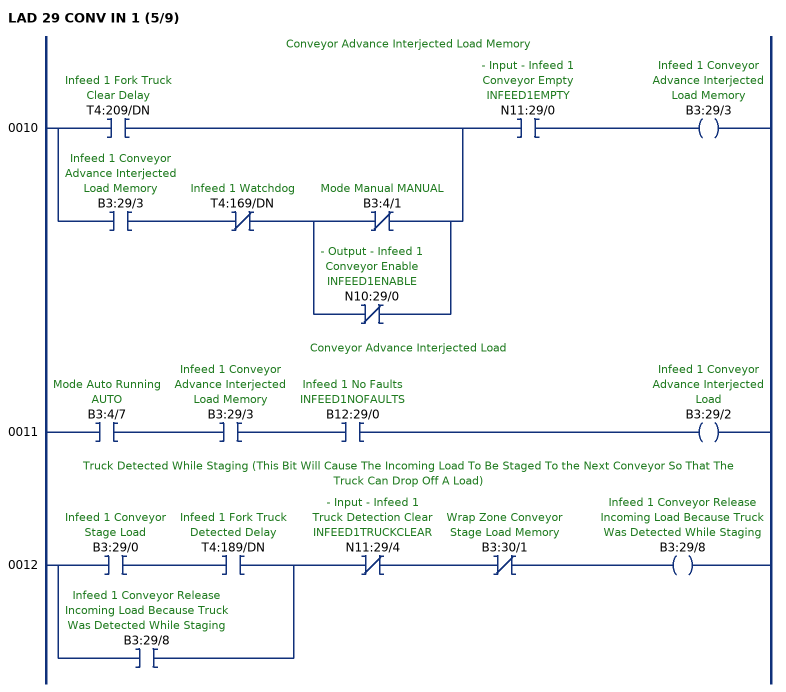
% Rung: 10 %
% Conveyor Advance Interjected Load Memory %
SOR BST XIC T4:209/DN NXB XIC B3:29/3 XIO T4:169/DN BST XIO B3:4/1 NXB XIO N10:29/0 BND BND XIC N11:29/0 OTE B3:29/3 EOR
%   T4:209  "Infeed 1 Fork Truck Clear Delay" %
%   B3:29/3  "Infeed 1 Conveyor Advance Interjected Load Memory" %
%   T4:169  "Infeed 1 Watchdog" %
%   B3:4/1  MANUAL  "Mode Manual" %
%   N10:29/0  INFEED1ENABLE  "- Output - Infeed 1 Conveyor Enable" %
%   N11:29/0  INFEED1EMPTY  "- Input - Infeed 1 Conveyor Empty" %
% Rung: 11 %
% Conveyor Advance Interjected Load %
SOR XIC B3:4/7 XIC B3:29/3 XIC B12:29/0 OTE B3:29/2 EOR
%   B3:4/7  AUTO  "Mode Auto Running" %
%   B3:29/3  "Infeed 1 Conveyor Advance Interjected Load Memory" %
%   B12:29/0  INFEED1NOFAULTS  "Infeed 1 No Faults" %
%   B3:29/2  "Infeed 1 Conveyor Advance Interjected Load" %
% Rung: 12 %
% Truck Detected While Staging (This Bit Will Cause The Incoming Load To Be Staged To the Next Conveyor So That The Truck Can Drop Off A Load) %
SOR BST XIC B3:29/0 XIC T4:189/DN NXB XIC B3:29/8 BND XIO N11:29/4 XIO B3:30/1 OTE B3:29/8 EOR
%   B3:29/0  "Infeed 1 Conveyor Stage Load" %
%   T4:189  "Infeed 1 Fork Truck Detected Delay" %
%   B3:29/8  "Infeed 1 Conveyor Release Incoming Load Because Truck Was Detected While Staging" %
%   N11:29/4  INFEED1TRUCKCLEAR  "- Input - Infeed 1 Truck Detection Clear" %
%   B3:30/1  "Wrap Zone Conveyor Stage Load Memory" %

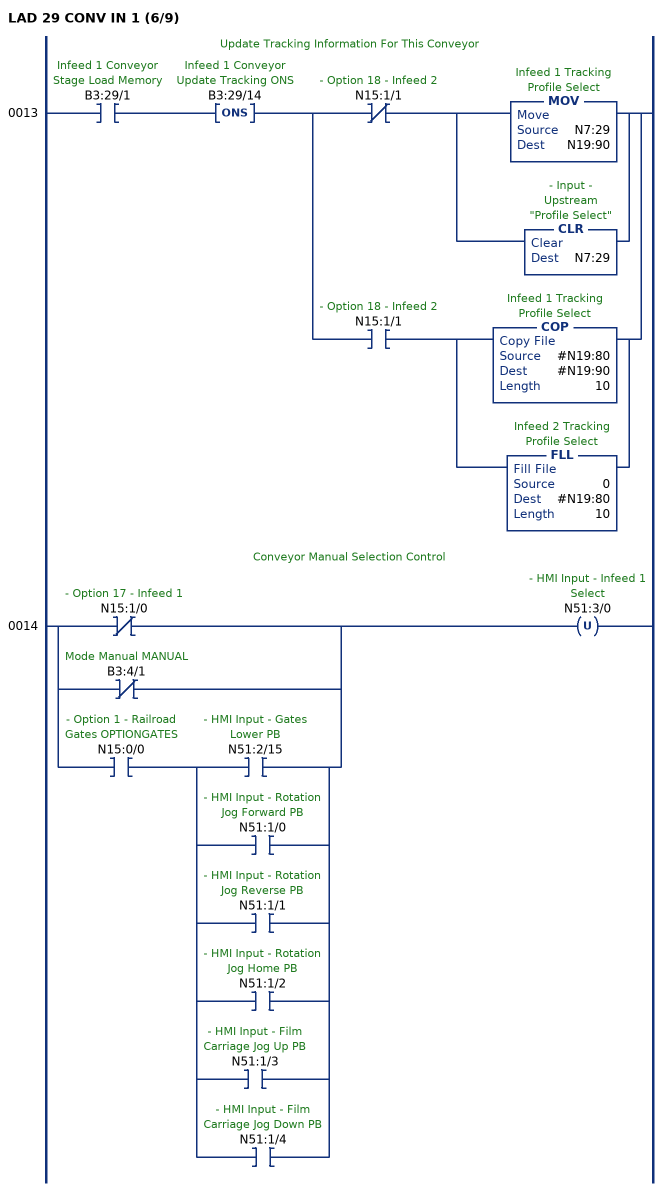
% Rung: 13 %
% Update Tracking Information For This Conveyor %
SOR XIC B3:29/1 ONS B3:29/14 BST XIO N15:1/1 BST MOV N7:29 N19:90 NXB CLR N7:29 BND NXB XIC N15:1/1 BST COP #N19:80 #N19:90 10 NXB FLL 0 #N19:80 10 BND BND EOR
%   B3:29/1  "Infeed 1 Conveyor Stage Load Memory" %
%   B3:29/14  "Infeed 1 Conveyor Update Tracking ONS" %
%   N15:1/1  "- Option 18 - Infeed 2" %
%   N7:29  "- Input - Upstream "Profile Select"" %
%   N19:90  "Infeed 1 Tracking Profile Select" %
%   N19:80  "Infeed 2 Tracking Profile Select" %
% Rung: 14 %
% Conveyor Manual Selection Control %
SOR BST XIO N15:1/0 NXB XIO B3:4/1 NXB XIC N15:0/0 BST XIC N51:2/15 NXB XIC N51:1/0 NXB XIC N51:1/1 NXB XIC N51:1/2 NXB XIC N51:1/3 NXB XIC N51:1/4 BND BND OTU N51:3/0 EOR
%   N15:1/0  "- Option 17 - Infeed 1" %
%   B3:4/1  MANUAL  "Mode Manual" %
%   N15:0/0  OPTIONGATES  "- Option 1 - Railroad Gates" %
%   N51:2/15  "- HMI Input - Gates Lower PB" %
%   N51:1/0  "- HMI Input - Rotation Jog Forward PB" %
%   N51:1/1  "- HMI Input - Rotation Jog Reverse PB" %
%   N51:1/2  "- HMI Input - Rotation Jog Home PB" %
%   N51:1/3  "- HMI Input - Film Carriage Jog Up PB" %
%   N51:1/4  "- HMI Input - Film Carriage Jog Down PB" %
%   N51:3/0  "- HMI Input - Infeed 1 Select" %

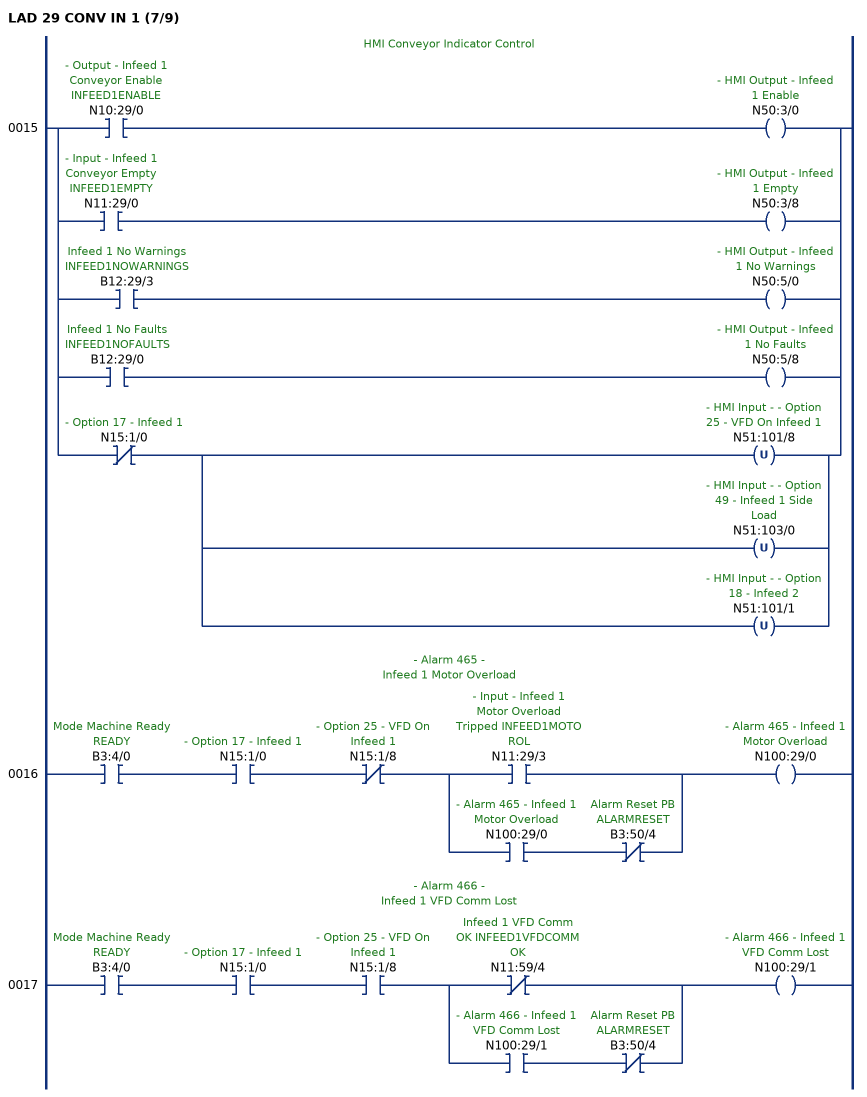
% Rung: 15 %
% HMI Conveyor Indicator Control %
SOR BST XIC N10:29/0 OTE N50:3/0 NXB XIC N11:29/0 OTE N50:3/8 NXB XIC B12:29/3 OTE N50:5/0 NXB XIC B12:29/0 OTE N50:5/8 NXB XIO N15:1/0 BST OTU N51:101/8 NXB OTU N51:103/0 NXB OTU N51:101/1 BND BND EOR
%   N10:29/0  INFEED1ENABLE  "- Output - Infeed 1 Conveyor Enable" %
%   N50:3/0  "- HMI Output - Infeed 1 Enable" %
%   N11:29/0  INFEED1EMPTY  "- Input - Infeed 1 Conveyor Empty" %
%   N50:3/8  "- HMI Output - Infeed 1 Empty" %
%   B12:29/3  INFEED1NOWARNINGS  "Infeed 1 No Warnings" %
%   N50:5/0  "- HMI Output - Infeed 1 No Warnings" %
%   B12:29/0  INFEED1NOFAULTS  "Infeed 1 No Faults" %
%   N50:5/8  "- HMI Output - Infeed 1 No Faults" %
%   N15:1/0  "- Option 17 - Infeed 1" %
%   N51:101/8  "- HMI Input - - Option 25 - VFD On Infeed 1" %
%   N51:103/0  "- HMI Input - - Option 49 - Infeed 1 Side Load" %
%   N51:101/1  "- HMI Input - - Option 18 - Infeed 2" %
% Rung: 16 %
% - Alarm 465 -
% 
% Infeed 1 Motor Overload %
SOR XIC B3:4/0 XIC N15:1/0 XIO N15:1/8 BST XIC N11:29/3 NXB XIC N100:29/0 XIO B3:50/4 BND OTE N100:29/0 EOR
%   B3:4/0  READY  "Mode Machine Ready" %
%   N15:1/0  "- Option 17 - Infeed 1" %
%   N15:1/8  "- Option 25 - VFD On Infeed 1" %
%   N11:29/3  INFEED1MOTOROL  "- Input - Infeed 1 Motor Overload Tripped" %
%   N100:29/0  "- Alarm 465 - Infeed 1 Motor Overload" %
%   B3:50/4  ALARMRESET  "Alarm Reset PB" %
% Rung: 17 %
% - Alarm 466 -
% 
% Infeed 1 VFD Comm Lost %
SOR XIC B3:4/0 XIC N15:1/0 XIC N15:1/8 BST XIO N11:59/4 NXB XIC N100:29/1 XIO B3:50/4 BND OTE N100:29/1 EOR
%   B3:4/0  READY  "Mode Machine Ready" %
%   N15:1/0  "- Option 17 - Infeed 1" %
%   N15:1/8  "- Option 25 - VFD On Infeed 1" %
%   N11:59/4  INFEED1VFDCOMMOK  "Infeed 1 VFD Comm OK" %
%   N100:29/1  "- Alarm 466 - Infeed 1 VFD Comm Lost" %
%   B3:50/4  ALARMRESET  "Alarm Reset PB" %

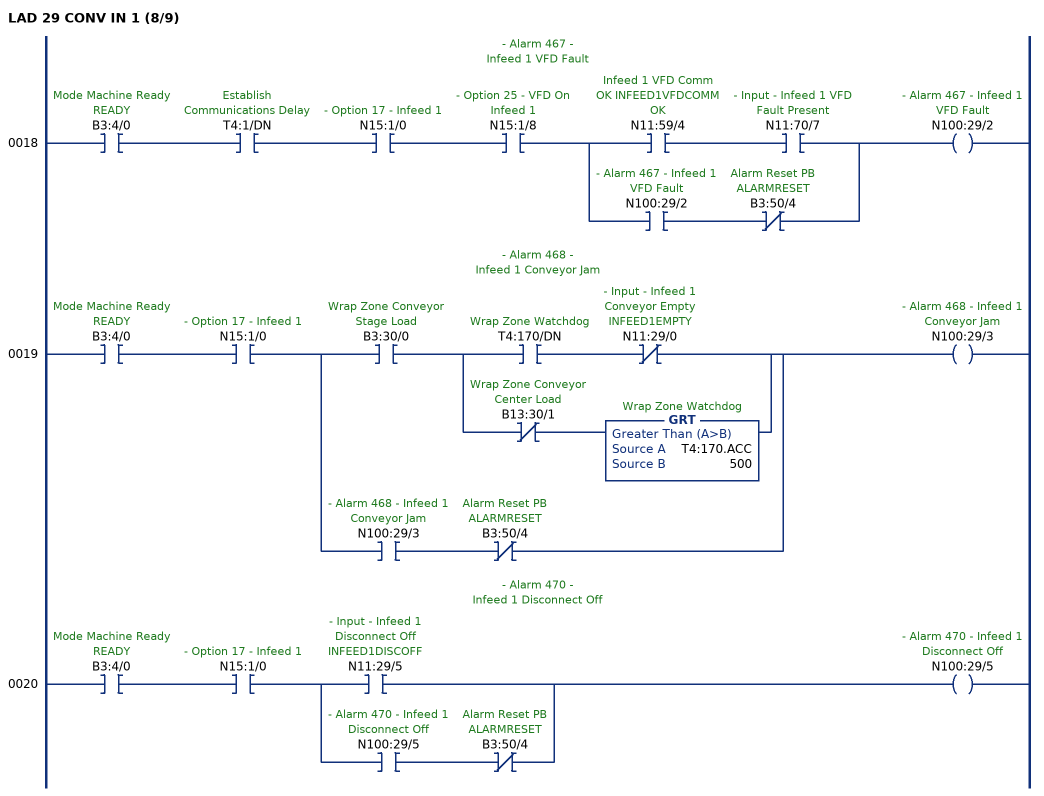
% Rung: 18 %
% - Alarm 467 -
% 
% Infeed 1 VFD Fault %
SOR XIC B3:4/0 XIC T4:1/DN XIC N15:1/0 XIC N15:1/8 BST XIC N11:59/4 XIC N11:70/7 NXB XIC N100:29/2 XIO B3:50/4 BND OTE N100:29/2 EOR
%   B3:4/0  READY  "Mode Machine Ready" %
%   T4:1  "Establish Communications Delay" %
%   N15:1/0  "- Option 17 - Infeed 1" %
%   N15:1/8  "- Option 25 - VFD On Infeed 1" %
%   N11:59/4  INFEED1VFDCOMMOK  "Infeed 1 VFD Comm OK" %
%   N11:70/7  "- Input - Infeed 1 VFD Fault Present" %
%   N100:29/2  "- Alarm 467 - Infeed 1 VFD Fault" %
%   B3:50/4  ALARMRESET  "Alarm Reset PB" %
% Rung: 19 %
% - Alarm 468 -
% 
% Infeed 1 Conveyor Jam %
SOR XIC B3:4/0 XIC N15:1/0 BST XIC B3:30/0 BST XIC T4:170/DN XIO N11:29/0 NXB XIO B13:30/1 GRT T4:170.ACC 500 BND NXB XIC N100:29/3 XIO B3:50/4 BND OTE N100:29/3 EOR
%   B3:4/0  READY  "Mode Machine Ready" %
%   N15:1/0  "- Option 17 - Infeed 1" %
%   B3:30/0  "Wrap Zone Conveyor Stage Load" %
%   T4:170  "Wrap Zone Watchdog" %
%   N11:29/0  INFEED1EMPTY  "- Input - Infeed 1 Conveyor Empty" %
%   B13:30/1  "Wrap Zone Conveyor Center Load" %
%   N100:29/3  "- Alarm 468 - Infeed 1 Conveyor Jam" %
%   B3:50/4  ALARMRESET  "Alarm Reset PB" %
% Rung: 20 %
% - Alarm 470 -
% 
% Infeed 1 Disconnect Off %
SOR XIC B3:4/0 XIC N15:1/0 BST XIC N11:29/5 NXB XIC N100:29/5 XIO B3:50/4 BND OTE N100:29/5 EOR
%   B3:4/0  READY  "Mode Machine Ready" %
%   N15:1/0  "- Option 17 - Infeed 1" %
%   N11:29/5  INFEED1DISCOFF  "- Input - Infeed 1 Disconnect Off" %
%   N100:29/5  "- Alarm 470 - Infeed 1 Disconnect Off" %
%   B3:50/4  ALARMRESET  "Alarm Reset PB" %

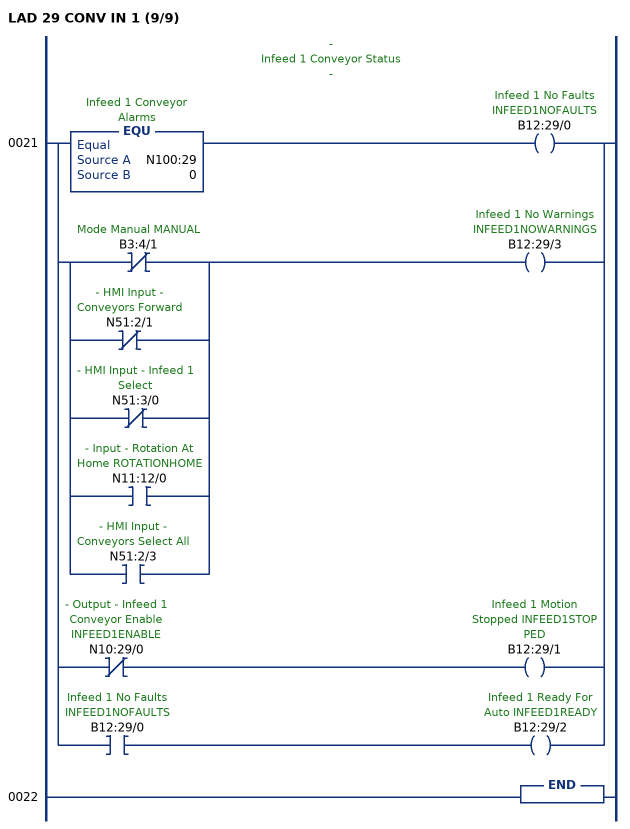
% Rung: 21 %
% -
% 
% Infeed 1 Conveyor Status
% 
% - %
SOR BST EQU N100:29 0 OTE B12:29/0 NXB BST XIO B3:4/1 NXB XIO N51:2/1 NXB XIO N51:3/0 NXB XIC N11:12/0 NXB XIC N51:2/3 BND OTE B12:29/3 NXB XIO N10:29/0 OTE B12:29/1 NXB XIC B12:29/0 OTE B12:29/2 BND EOR
%   N100:29  "Infeed 1 Conveyor Alarms" %
%   B12:29/0  INFEED1NOFAULTS  "Infeed 1 No Faults" %
%   B3:4/1  MANUAL  "Mode Manual" %
%   N51:2/1  "- HMI Input - Conveyors Forward" %
%   N51:3/0  "- HMI Input - Infeed 1 Select" %
%   N11:12/0  ROTATIONHOME  "- Input - Rotation At Home" %
%   N51:2/3  "- HMI Input - Conveyors Select All" %
%   B12:29/3  INFEED1NOWARNINGS  "Infeed 1 No Warnings" %
%   N10:29/0  INFEED1ENABLE  "- Output - Infeed 1 Conveyor Enable" %
%   B12:29/1  INFEED1STOPPED  "Infeed 1 Motion Stopped" %
%   B12:29/2  INFEED1READY  "Infeed 1 Ready For Auto" %
% Rung: 22 %
SOR END EOR

LADDER 30 "CONV WRAPZ"
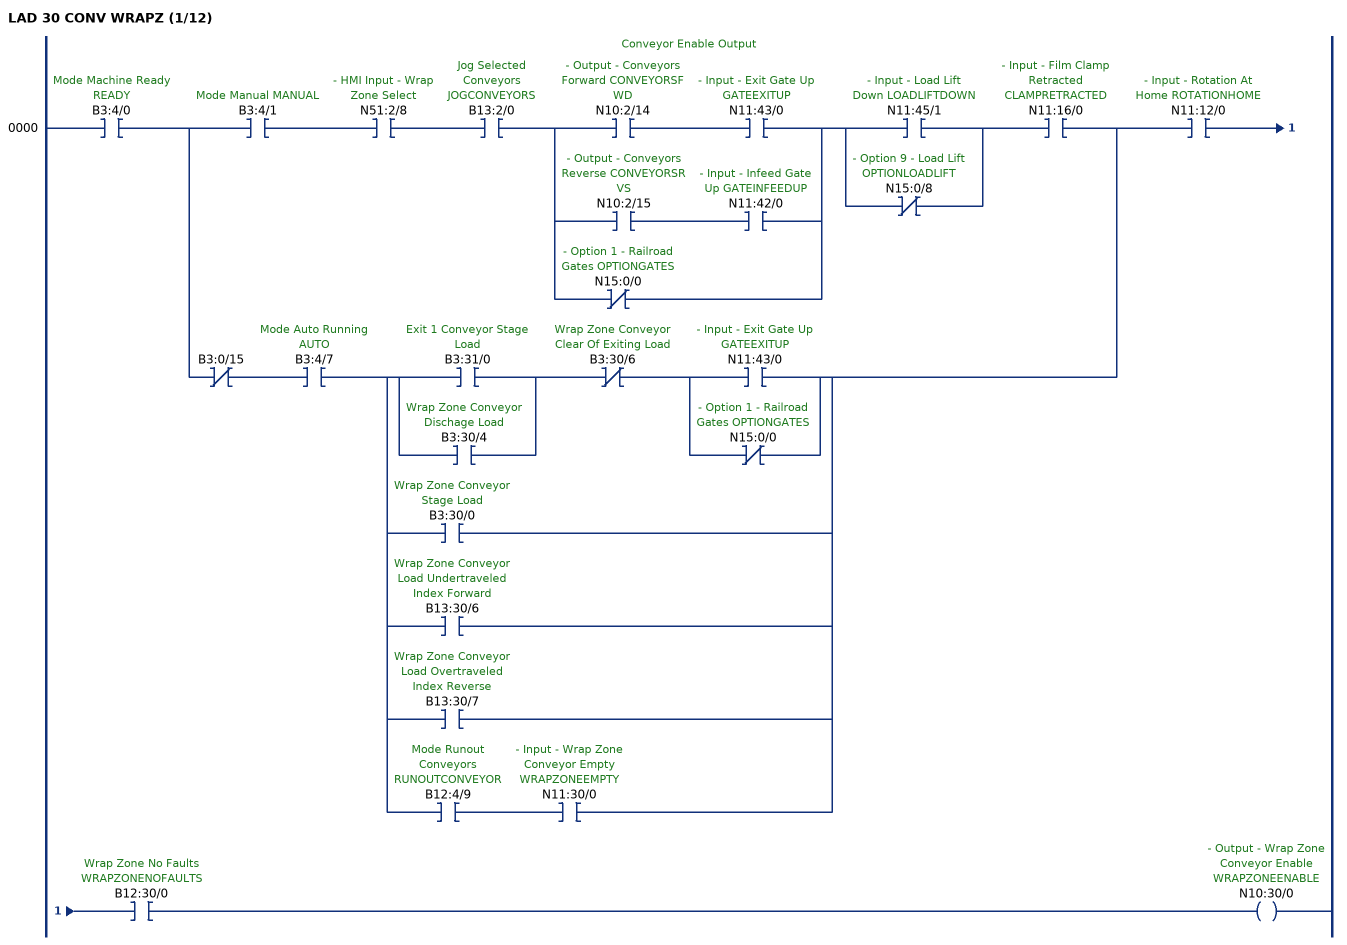
% Rung: 0 %
% Conveyor Enable Output %
SOR XIC B3:4/0 BST XIC B3:4/1 XIC N51:2/8 XIC B13:2/0 BST XIC N10:2/14 XIC N11:43/0 NXB XIC N10:2/15 XIC N11:42/0 NXB XIO N15:0/0 BND BST XIC N11:45/1 NXB XIO N15:0/8 BND XIC N11:16/0 NXB XIO B3:0/15 XIC B3:4/7 BST BST XIC B3:31/0 NXB XIC B3:30/4 BND XIO B3:30/6 BST XIC N11:43/0 NXB XIO N15:0/0 BND NXB XIC B3:30/0 NXB XIC B13:30/6 NXB XIC B13:30/7 NXB XIC B12:4/9 XIC N11:30/0 BND BND XIC N11:12/0 XIC B12:30/0 OTE N10:30/0 EOR
%   B3:4/0  READY  "Mode Machine Ready" %
%   B3:4/1  MANUAL  "Mode Manual" %
%   N51:2/8  "- HMI Input - Wrap Zone Select" %
%   B13:2/0  JOGCONVEYORS  "Jog Selected Conveyors" %
%   N10:2/14  CONVEYORSFWD  "- Output - Conveyors Forward" %
%   N11:43/0  GATEEXITUP  "- Input - Exit Gate Up" %
%   N10:2/15  CONVEYORSRVS  "- Output - Conveyors Reverse" %
%   N11:42/0  GATEINFEEDUP  "- Input - Infeed Gate Up" %
%   N15:0/0  OPTIONGATES  "- Option 1 - Railroad Gates" %
%   N11:45/1  LOADLIFTDOWN  "- Input - Load Lift Down" %
%   N15:0/8  OPTIONLOADLIFT  "- Option 9 - Load Lift" %
%   N11:16/0  CLAMPRETRACTED  "- Input - Film Clamp Retracted" %
%   B3:4/7  AUTO  "Mode Auto Running" %
%   B3:31/0  "Exit 1 Conveyor Stage Load" %
%   B3:30/4  "Wrap Zone Conveyor Dischage Load" %
%   B3:30/6  "Wrap Zone Conveyor Clear Of Exiting Load" %
%   B3:30/0  "Wrap Zone Conveyor Stage Load" %
%   B13:30/6  "Wrap Zone Conveyor Load Undertraveled Index Forward" %
%   B13:30/7  "Wrap Zone Conveyor Load Overtraveled Index Reverse" %
%   B12:4/9  RUNOUTCONVEYOR  "Mode Runout Conveyors" %
%   N11:30/0  WRAPZONEEMPTY  "- Input - Wrap Zone Conveyor Empty" %
%   N11:12/0  ROTATIONHOME  "- Input - Rotation At Home" %
%   B12:30/0  WRAPZONENOFAULTS  "Wrap Zone No Faults" %
%   N10:30/0  WRAPZONEENABLE  "- Output - Wrap Zone Conveyor Enable" %

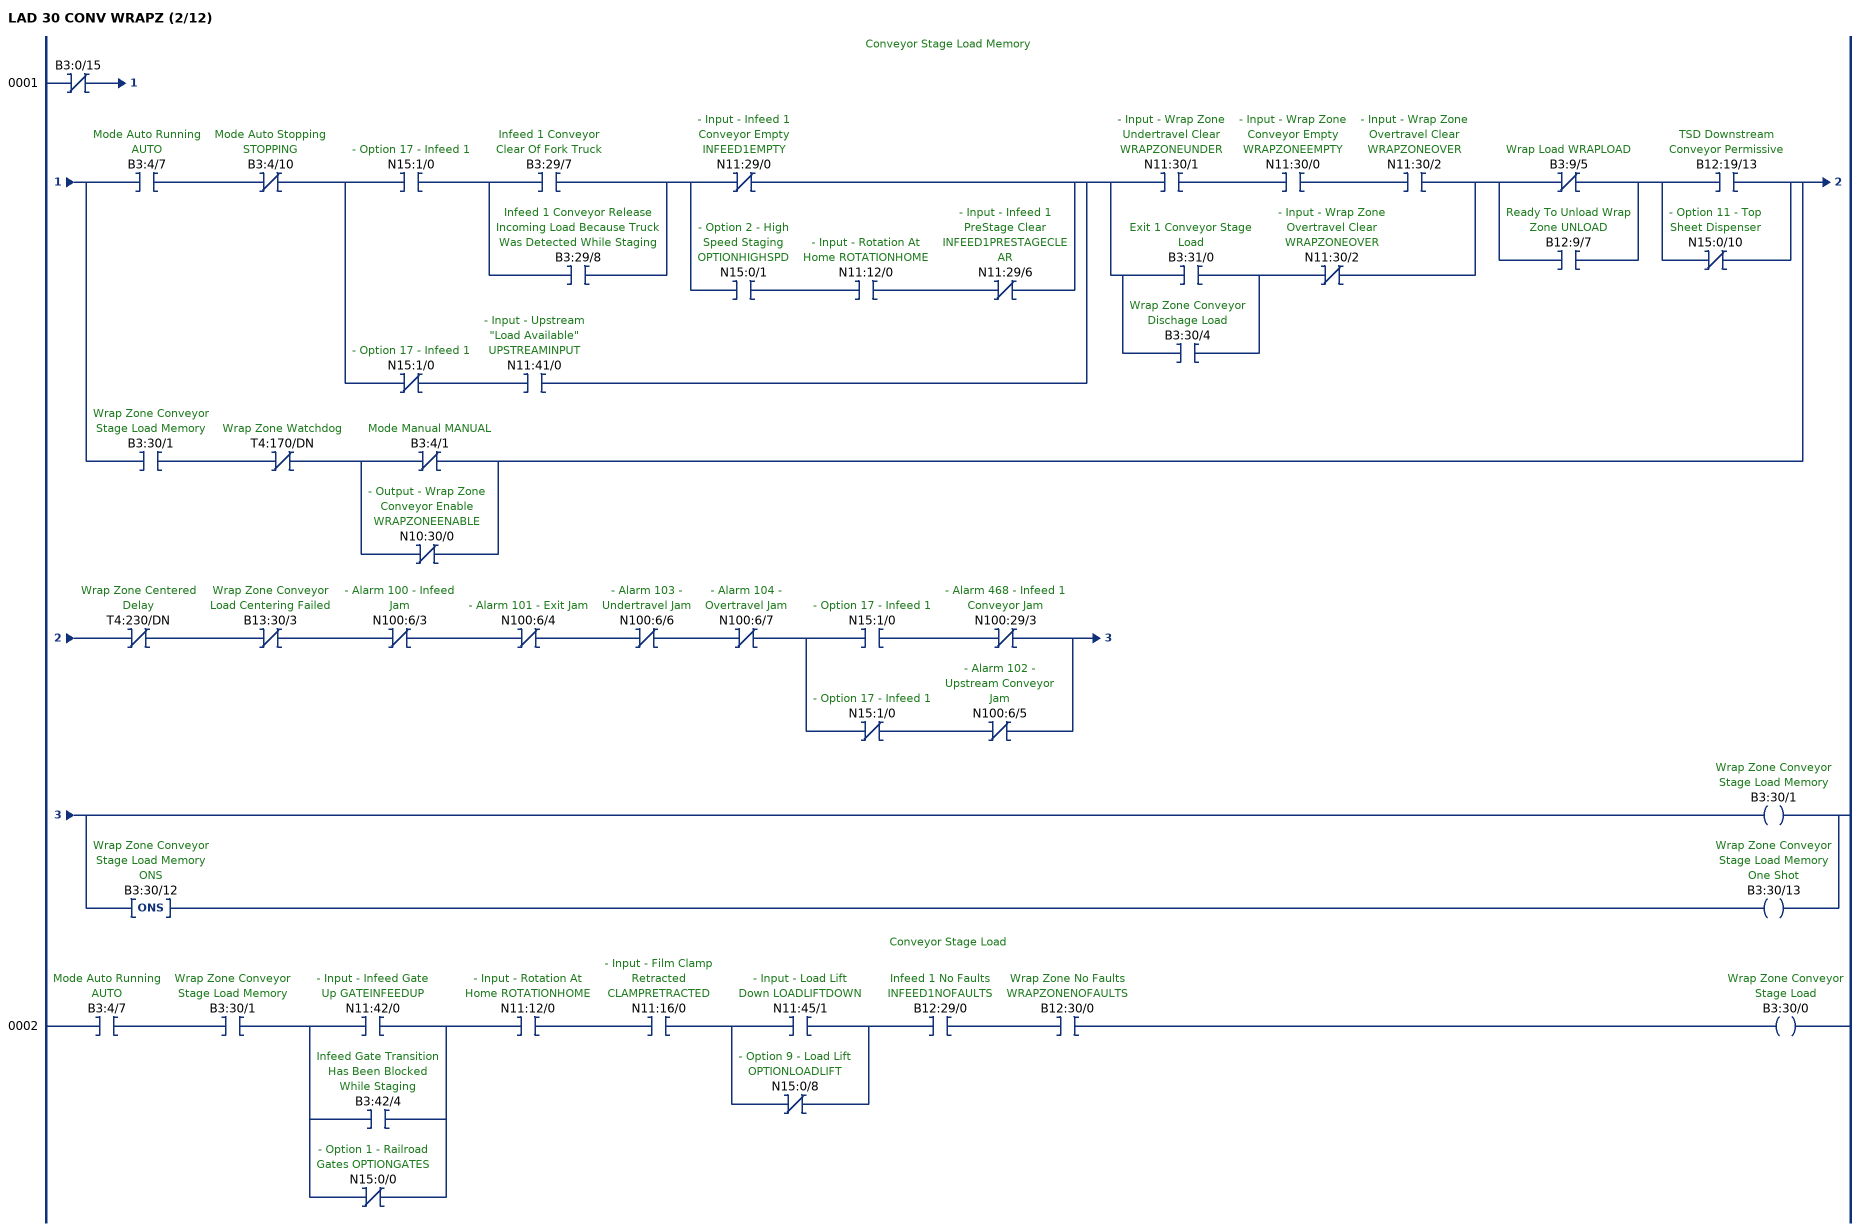
% Rung: 1 %
% Conveyor Stage Load Memory %
SOR XIO B3:0/15 BST XIC B3:4/7 XIO B3:4/10 BST XIC N15:1/0 BST XIC B3:29/7 NXB XIC B3:29/8 BND BST XIO N11:29/0 NXB XIC N15:0/1 XIC N11:12/0 XIO N11:29/6 BND NXB XIO N15:1/0 XIC N11:41/0 BND BST XIC N11:30/1 XIC N11:30/0 XIC N11:30/2 NXB BST XIC B3:31/0 NXB XIC B3:30/4 BND XIO N11:30/2 BND BST XIO B3:9/5 NXB XIC B12:9/7 BND BST XIC B12:19/13 NXB XIO N15:0/10 BND NXB XIC B3:30/1 XIO T4:170/DN BST XIO B3:4/1 NXB XIO N10:30/0 BND BND XIO T4:230/DN XIO B13:30/3 XIO N100:6/3 XIO N100:6/4 XIO N100:6/6 XIO N100:6/7 BST XIC N15:1/0 XIO N100:29/3 NXB XIO N15:1/0 XIO N100:6/5 BND BST OTE B3:30/1 NXB ONS B3:30/12 OTE B3:30/13 BND EOR
%   B3:4/7  AUTO  "Mode Auto Running" %
%   B3:4/10  STOPPING  "Mode Auto Stopping" %
%   N15:1/0  "- Option 17 - Infeed 1" %
%   B3:29/7  "Infeed 1 Conveyor Clear Of Fork Truck" %
%   B3:29/8  "Infeed 1 Conveyor Release Incoming Load Because Truck Was Detected While Staging" %
%   N11:29/0  INFEED1EMPTY  "- Input - Infeed 1 Conveyor Empty" %
%   N15:0/1  OPTIONHIGHSPD  "- Option 2 - High Speed Staging" %
%   N11:12/0  ROTATIONHOME  "- Input - Rotation At Home" %
%   N11:29/6  INFEED1PRESTAGECLEAR  "- Input - Infeed 1 PreStage Clear" %
%   N11:41/0  UPSTREAMINPUT  "- Input - Upstream "Load Available"" %
%   N11:30/1  WRAPZONEUNDER  "- Input - Wrap Zone Undertravel Clear" %
%   N11:30/0  WRAPZONEEMPTY  "- Input - Wrap Zone Conveyor Empty" %
%   N11:30/2  WRAPZONEOVER  "- Input - Wrap Zone Overtravel Clear" %
%   B3:31/0  "Exit 1 Conveyor Stage Load" %
%   B3:30/4  "Wrap Zone Conveyor Dischage Load" %
%   B3:9/5  WRAPLOAD  "Wrap Load" %
%   B12:9/7  UNLOAD  "Ready To Unload Wrap Zone" %
%   B12:19/13  "TSD Downstream Conveyor Permissive" %
%   N15:0/10  "- Option 11 - Top Sheet Dispenser" %
%   B3:30/1  "Wrap Zone Conveyor Stage Load Memory" %
%   T4:170  "Wrap Zone Watchdog" %
%   B3:4/1  MANUAL  "Mode Manual" %
%   N10:30/0  WRAPZONEENABLE  "- Output - Wrap Zone Conveyor Enable" %
%   T4:230  "Wrap Zone Centered Delay" %
%   B13:30/3  "Wrap Zone Conveyor Load Centering Failed" %
%   N100:6/3  "- Alarm 100 - Infeed Jam" %
%   N100:6/4  "- Alarm 101 - Exit Jam" %
%   N100:6/6  "- Alarm 103 - Undertravel Jam" %
%   N100:6/7  "- Alarm 104 - Overtravel Jam" %
%   N100:29/3  "- Alarm 468 - Infeed 1 Conveyor Jam" %
%   N100:6/5  "- Alarm 102 - Upstream Conveyor Jam" %
%   B3:30/12  "Wrap Zone Conveyor Stage Load Memory ONS" %
%   B3:30/13  "Wrap Zone Conveyor Stage Load Memory One Shot" %
% Rung: 2 %
% Conveyor Stage Load %
SOR XIC B3:4/7 XIC B3:30/1 BST XIC N11:42/0 NXB XIC B3:42/4 NXB XIO N15:0/0 BND XIC N11:12/0 XIC N11:16/0 BST XIC N11:45/1 NXB XIO N15:0/8 BND XIC B12:29/0 XIC B12:30/0 OTE B3:30/0 EOR
%   B3:4/7  AUTO  "Mode Auto Running" %
%   B3:30/1  "Wrap Zone Conveyor Stage Load Memory" %
%   N11:42/0  GATEINFEEDUP  "- Input - Infeed Gate Up" %
%   B3:42/4  "Infeed Gate Transition Has Been Blocked While Staging" %
%   N15:0/0  OPTIONGATES  "- Option 1 - Railroad Gates" %
%   N11:12/0  ROTATIONHOME  "- Input - Rotation At Home" %
%   N11:16/0  CLAMPRETRACTED  "- Input - Film Clamp Retracted" %
%   N11:45/1  LOADLIFTDOWN  "- Input - Load Lift Down" %
%   N15:0/8  OPTIONLOADLIFT  "- Option 9 - Load Lift" %
%   B12:29/0  INFEED1NOFAULTS  "Infeed 1 No Faults" %
%   B12:30/0  WRAPZONENOFAULTS  "Wrap Zone No Faults" %
%   B3:30/0  "Wrap Zone Conveyor Stage Load" %

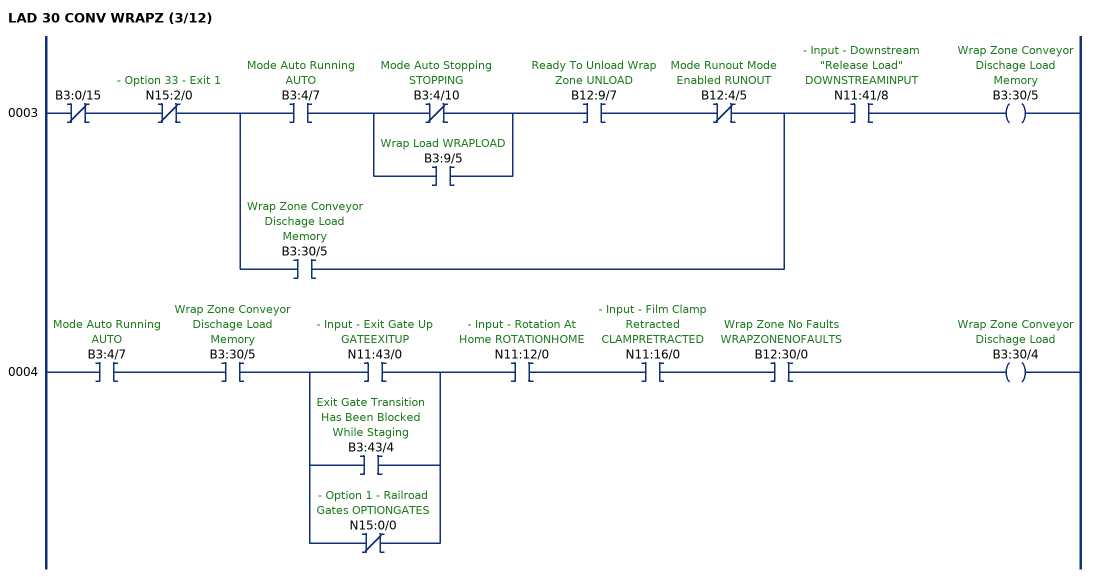
% Rung: 3 %
SOR XIO B3:0/15 XIO N15:2/0 BST XIC B3:4/7 BST XIO B3:4/10 NXB XIC B3:9/5 BND XIC B12:9/7 XIO B12:4/5 NXB XIC B3:30/5 BND XIC N11:41/8 OTE B3:30/5 EOR
%   N15:2/0  "- Option 33 - Exit 1" %
%   B3:4/7  AUTO  "Mode Auto Running" %
%   B3:4/10  STOPPING  "Mode Auto Stopping" %
%   B3:9/5  WRAPLOAD  "Wrap Load" %
%   B12:9/7  UNLOAD  "Ready To Unload Wrap Zone" %
%   B12:4/5  RUNOUT  "Mode Runout Mode Enabled" %
%   B3:30/5  "Wrap Zone Conveyor Dischage Load Memory" %
%   N11:41/8  DOWNSTREAMINPUT  "- Input - Downstream "Release Load"" %
% Rung: 4 %
SOR XIC B3:4/7 XIC B3:30/5 BST XIC N11:43/0 NXB XIC B3:43/4 NXB XIO N15:0/0 BND XIC N11:12/0 XIC N11:16/0 XIC B12:30/0 OTE B3:30/4 EOR
%   B3:4/7  AUTO  "Mode Auto Running" %
%   B3:30/5  "Wrap Zone Conveyor Dischage Load Memory" %
%   N11:43/0  GATEEXITUP  "- Input - Exit Gate Up" %
%   B3:43/4  "Exit Gate Transition Has Been Blocked While Staging" %
%   N15:0/0  OPTIONGATES  "- Option 1 - Railroad Gates" %
%   N11:12/0  ROTATIONHOME  "- Input - Rotation At Home" %
%   N11:16/0  CLAMPRETRACTED  "- Input - Film Clamp Retracted" %
%   B12:30/0  WRAPZONENOFAULTS  "Wrap Zone No Faults" %
%   B3:30/4  "Wrap Zone Conveyor Dischage Load" %

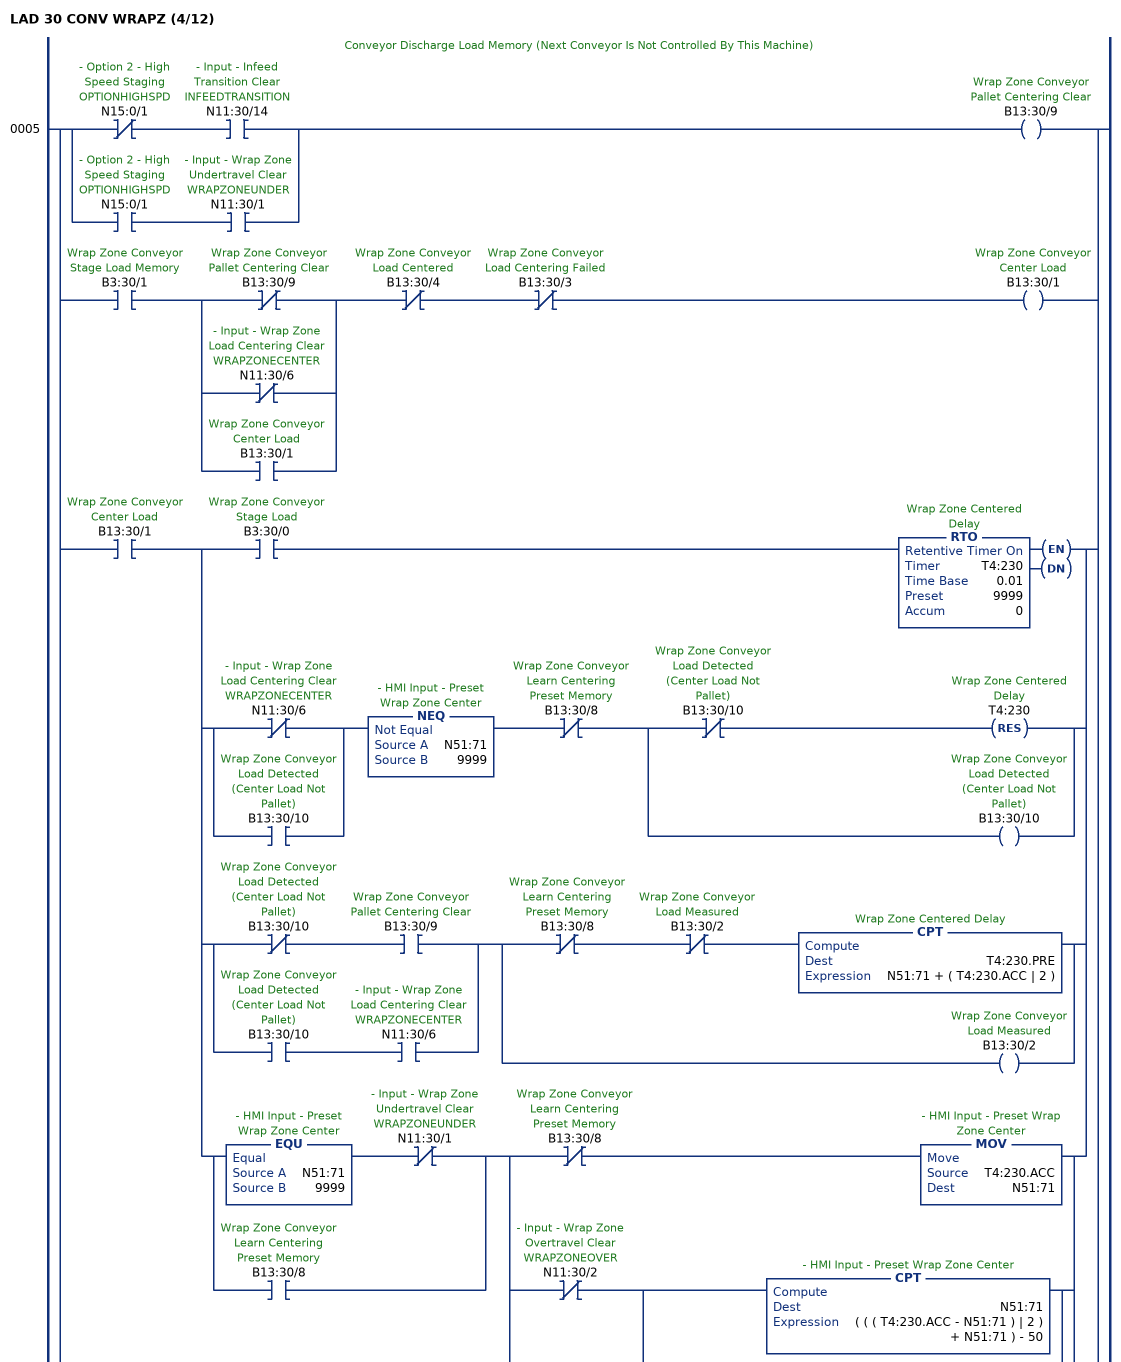

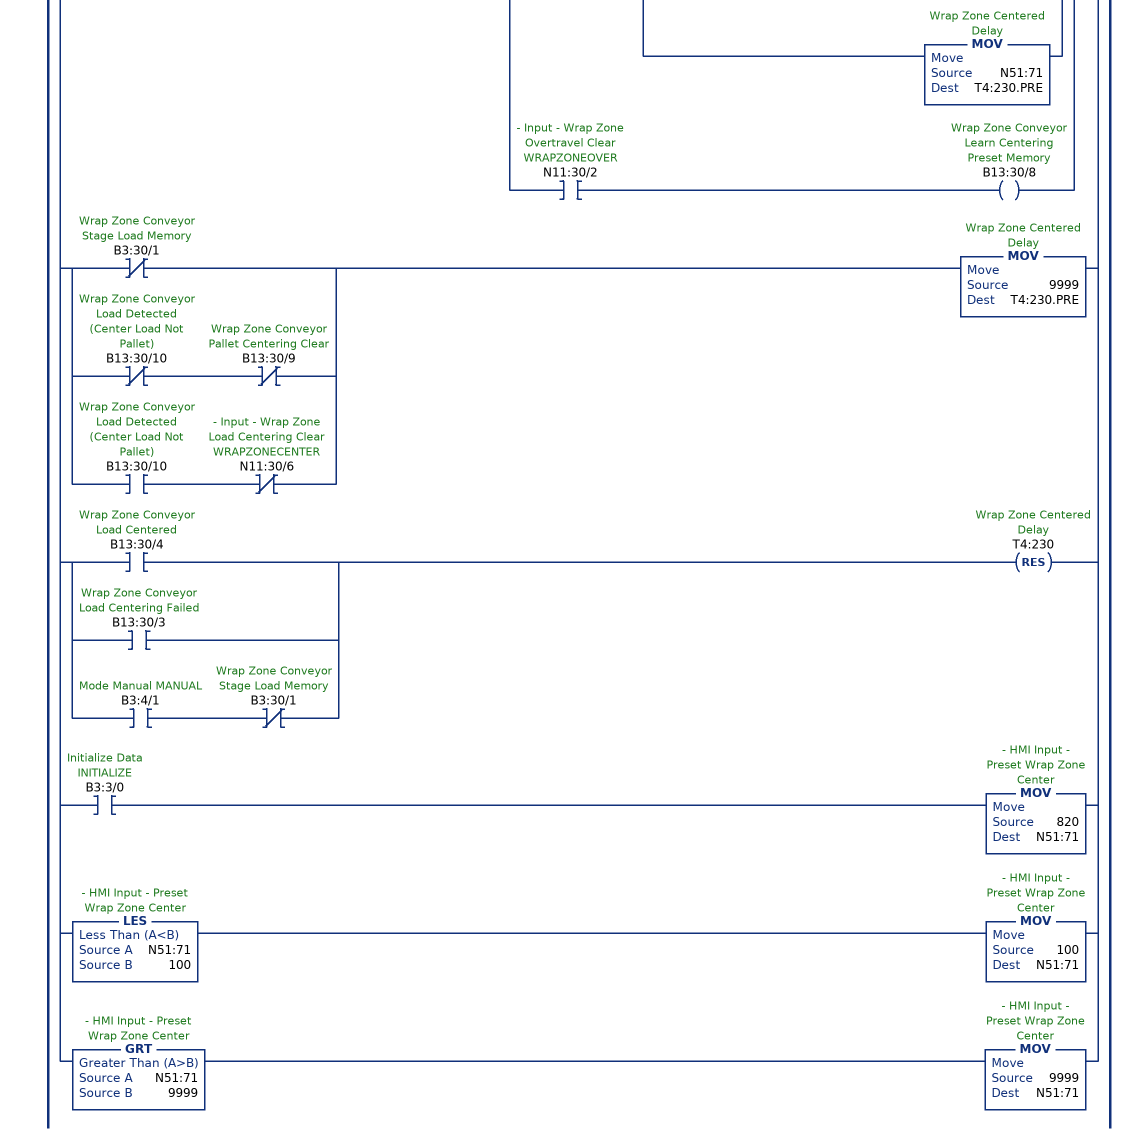
% Rung: 5 %
% Conveyor Discharge Load Memory (Next Conveyor Is Not Controlled By This Machine) %
SOR BST BST XIO N15:0/1 XIC N11:30/14 NXB XIC N15:0/1 XIC N11:30/1 BND OTE B13:30/9 NXB XIC B3:30/1 BST XIO B13:30/9 NXB XIO N11:30/6 NXB XIC B13:30/1 BND XIO B13:30/4 XIO B13:30/3 OTE B13:30/1 NXB XIC B13:30/1 BST XIC B3:30/0 RTO T4:230 0.01 9999 0 NXB BST XIO N11:30/6 NXB XIC B13:30/10 BND NEQ N51:71 9999 XIO B13:30/8 BST XIO B13:30/10 RES T4:230 NXB OTE B13:30/10 BND NXB BST XIO B13:30/10 XIC B13:30/9 NXB XIC B13:30/10 XIC N11:30/6 BND BST XIO B13:30/8 XIO B13:30/2 CPT T4:230.PRE " N51:71 + ( T4:230.ACC | 2 ) " NXB OTE B13:30/2 BND NXB BST EQU N51:71 9999 XIO N11:30/1 NXB XIC B13:30/8 BND BST XIO B13:30/8 MOV T4:230.ACC N51:71 NXB XIO N11:30/2 BST CPT N51:71 " ( ( ( T4:230.ACC - N51:71 ) | 2 ) + N51:71 ) - 50 " NXB MOV N51:71 T4:230.PRE BND NXB XIC N11:30/2 OTE B13:30/8 BND BND NXB BST XIO B3:30/1 NXB XIO B13:30/10 XIO B13:30/9 NXB XIC B13:30/10 XIO N11:30/6 BND MOV 9999 T4:230.PRE NXB BST XIC B13:30/4 NXB XIC B13:30/3 NXB XIC B3:4/1 XIO B3:30/1 BND RES T4:230 NXB BST XIC B3:3/0 MOV 820 N51:71 NXB LES N51:71 100 MOV 100 N51:71 NXB GRT N51:71 9999 MOV 9999 N51:71 BND BND EOR
%   N15:0/1  OPTIONHIGHSPD  "- Option 2 - High Speed Staging" %
%   N11:30/14  INFEEDTRANSITION  "- Input - Infeed Transition Clear" %
%   N11:30/1  WRAPZONEUNDER  "- Input - Wrap Zone Undertravel Clear" %
%   B13:30/9  "Wrap Zone Conveyor Pallet Centering Clear" %
%   B3:30/1  "Wrap Zone Conveyor Stage Load Memory" %
%   N11:30/6  WRAPZONECENTER  "- Input - Wrap Zone Load Centering Clear" %
%   B13:30/1  "Wrap Zone Conveyor Center Load" %
%   B13:30/4  "Wrap Zone Conveyor Load Centered" %
%   B13:30/3  "Wrap Zone Conveyor Load Centering Failed" %
%   B3:30/0  "Wrap Zone Conveyor Stage Load" %
%   T4:230  "Wrap Zone Centered Delay" %
%   B13:30/10  "Wrap Zone Conveyor Load Detected (Center Load Not Pallet)" %
%   N51:71  "- HMI Input - Preset Wrap Zone Center" %
%   B13:30/8  "Wrap Zone Conveyor Learn Centering Preset Memory" %
%   B13:30/2  "Wrap Zone Conveyor Load Measured" %
%   N11:30/2  WRAPZONEOVER  "- Input - Wrap Zone Overtravel Clear" %
%   B3:4/1  MANUAL  "Mode Manual" %
%   B3:3/0  INITIALIZE  "Initialize Data" %

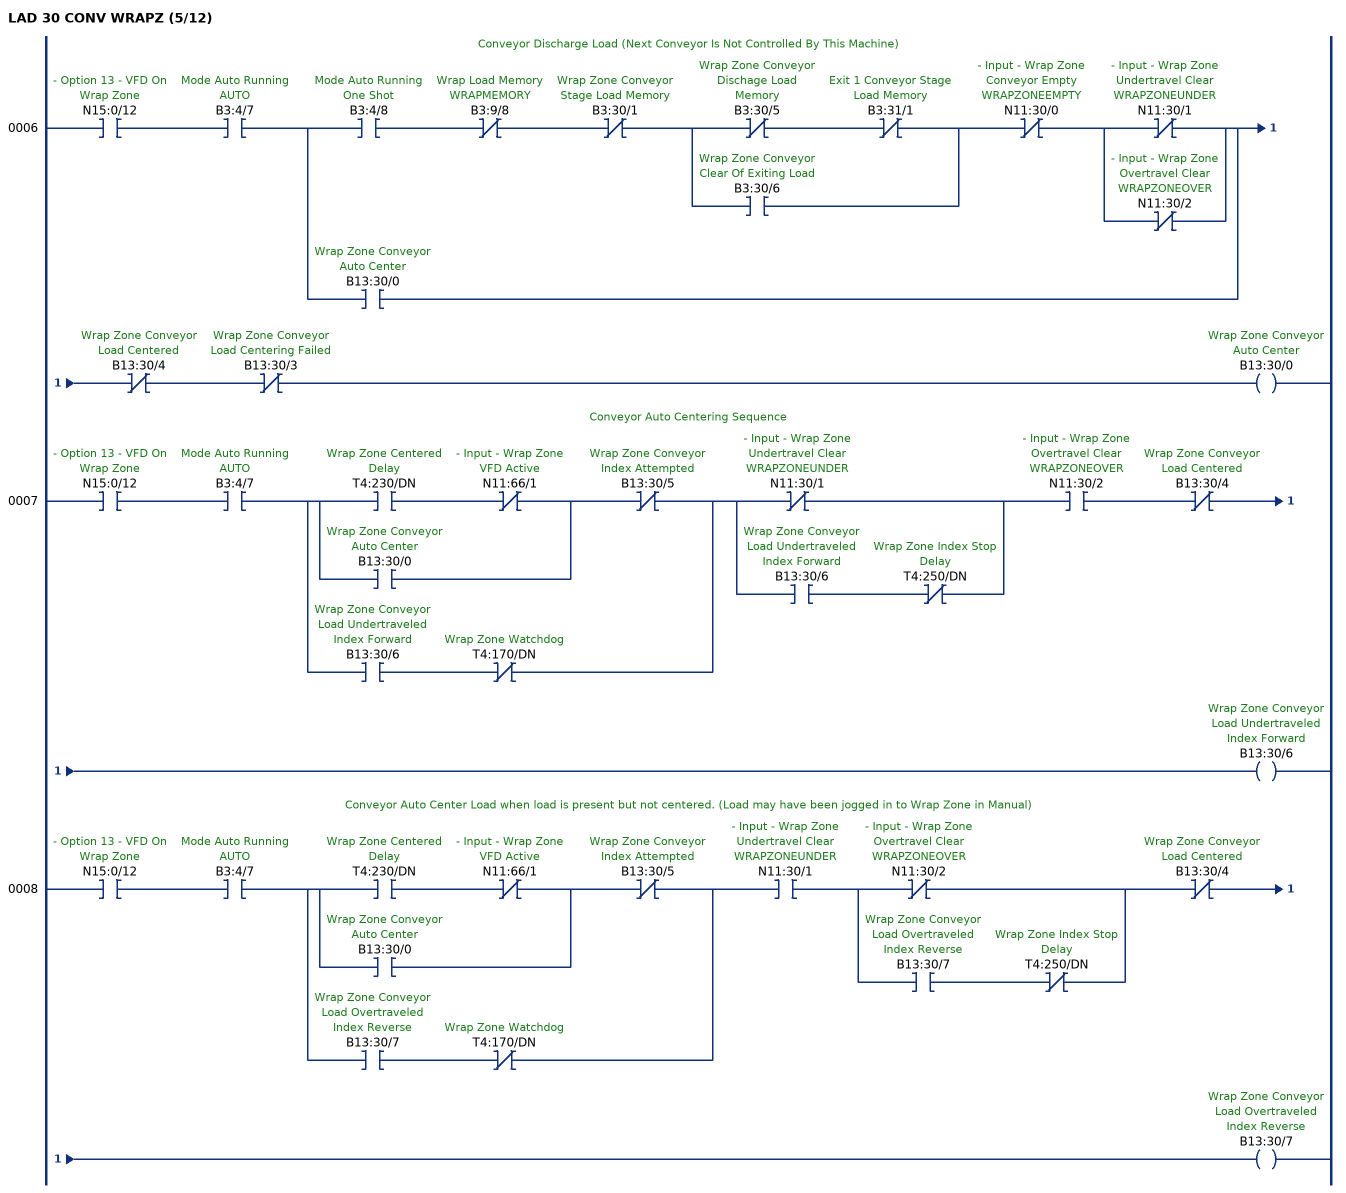
% Rung: 6 %
% Conveyor Discharge Load (Next Conveyor Is Not Controlled By This Machine) %
SOR XIC N15:0/12 XIC B3:4/7 BST XIC B3:4/8 XIO B3:9/8 XIO B3:30/1 BST XIO B3:30/5 XIO B3:31/1 NXB XIC B3:30/6 BND XIO N11:30/0 BST XIO N11:30/1 NXB XIO N11:30/2 BND NXB XIC B13:30/0 BND XIO B13:30/4 XIO B13:30/3 OTE B13:30/0 EOR
%   N15:0/12  "- Option 13 - VFD On Wrap Zone" %
%   B3:4/7  AUTO  "Mode Auto Running" %
%   B3:4/8  "Mode Auto Running One Shot" %
%   B3:9/8  WRAPMEMORY  "Wrap Load Memory" %
%   B3:30/1  "Wrap Zone Conveyor Stage Load Memory" %
%   B3:30/5  "Wrap Zone Conveyor Dischage Load Memory" %
%   B3:31/1  "Exit 1 Conveyor Stage Load Memory" %
%   B3:30/6  "Wrap Zone Conveyor Clear Of Exiting Load" %
%   N11:30/0  WRAPZONEEMPTY  "- Input - Wrap Zone Conveyor Empty" %
%   N11:30/1  WRAPZONEUNDER  "- Input - Wrap Zone Undertravel Clear" %
%   N11:30/2  WRAPZONEOVER  "- Input - Wrap Zone Overtravel Clear" %
%   B13:30/0  "Wrap Zone Conveyor Auto Center" %
%   B13:30/4  "Wrap Zone Conveyor Load Centered" %
%   B13:30/3  "Wrap Zone Conveyor Load Centering Failed" %
% Rung: 7 %
% Conveyor Auto Centering Sequence %
SOR XIC N15:0/12 XIC B3:4/7 BST BST XIC T4:230/DN XIO N11:66/1 NXB XIC B13:30/0 BND XIO B13:30/5 NXB XIC B13:30/6 XIO T4:170/DN BND BST XIO N11:30/1 NXB XIC B13:30/6 XIO T4:250/DN BND XIC N11:30/2 XIO B13:30/4 OTE B13:30/6 EOR
%   N15:0/12  "- Option 13 - VFD On Wrap Zone" %
%   B3:4/7  AUTO  "Mode Auto Running" %
%   T4:230  "Wrap Zone Centered Delay" %
%   N11:66/1  "- Input - Wrap Zone VFD Active" %
%   B13:30/0  "Wrap Zone Conveyor Auto Center" %
%   B13:30/5  "Wrap Zone Conveyor Index Attempted" %
%   B13:30/6  "Wrap Zone Conveyor Load Undertraveled Index Forward" %
%   T4:170  "Wrap Zone Watchdog" %
%   N11:30/1  WRAPZONEUNDER  "- Input - Wrap Zone Undertravel Clear" %
%   T4:250  "Wrap Zone Index Stop Delay" %
%   N11:30/2  WRAPZONEOVER  "- Input - Wrap Zone Overtravel Clear" %
%   B13:30/4  "Wrap Zone Conveyor Load Centered" %
% Rung: 8 %
% Conveyor Auto Center Load when load is present but not centered. (Load may have been jogged in to Wrap Zone in Manual) %
SOR XIC N15:0/12 XIC B3:4/7 BST BST XIC T4:230/DN XIO N11:66/1 NXB XIC B13:30/0 BND XIO B13:30/5 NXB XIC B13:30/7 XIO T4:170/DN BND XIC N11:30/1 BST XIO N11:30/2 NXB XIC B13:30/7 XIO T4:250/DN BND XIO B13:30/4 OTE B13:30/7 EOR
%   N15:0/12  "- Option 13 - VFD On Wrap Zone" %
%   B3:4/7  AUTO  "Mode Auto Running" %
%   T4:230  "Wrap Zone Centered Delay" %
%   N11:66/1  "- Input - Wrap Zone VFD Active" %
%   B13:30/0  "Wrap Zone Conveyor Auto Center" %
%   B13:30/5  "Wrap Zone Conveyor Index Attempted" %
%   B13:30/7  "Wrap Zone Conveyor Load Overtraveled Index Reverse" %
%   T4:170  "Wrap Zone Watchdog" %
%   N11:30/1  WRAPZONEUNDER  "- Input - Wrap Zone Undertravel Clear" %
%   N11:30/2  WRAPZONEOVER  "- Input - Wrap Zone Overtravel Clear" %
%   T4:250  "Wrap Zone Index Stop Delay" %
%   B13:30/4  "Wrap Zone Conveyor Load Centered" %

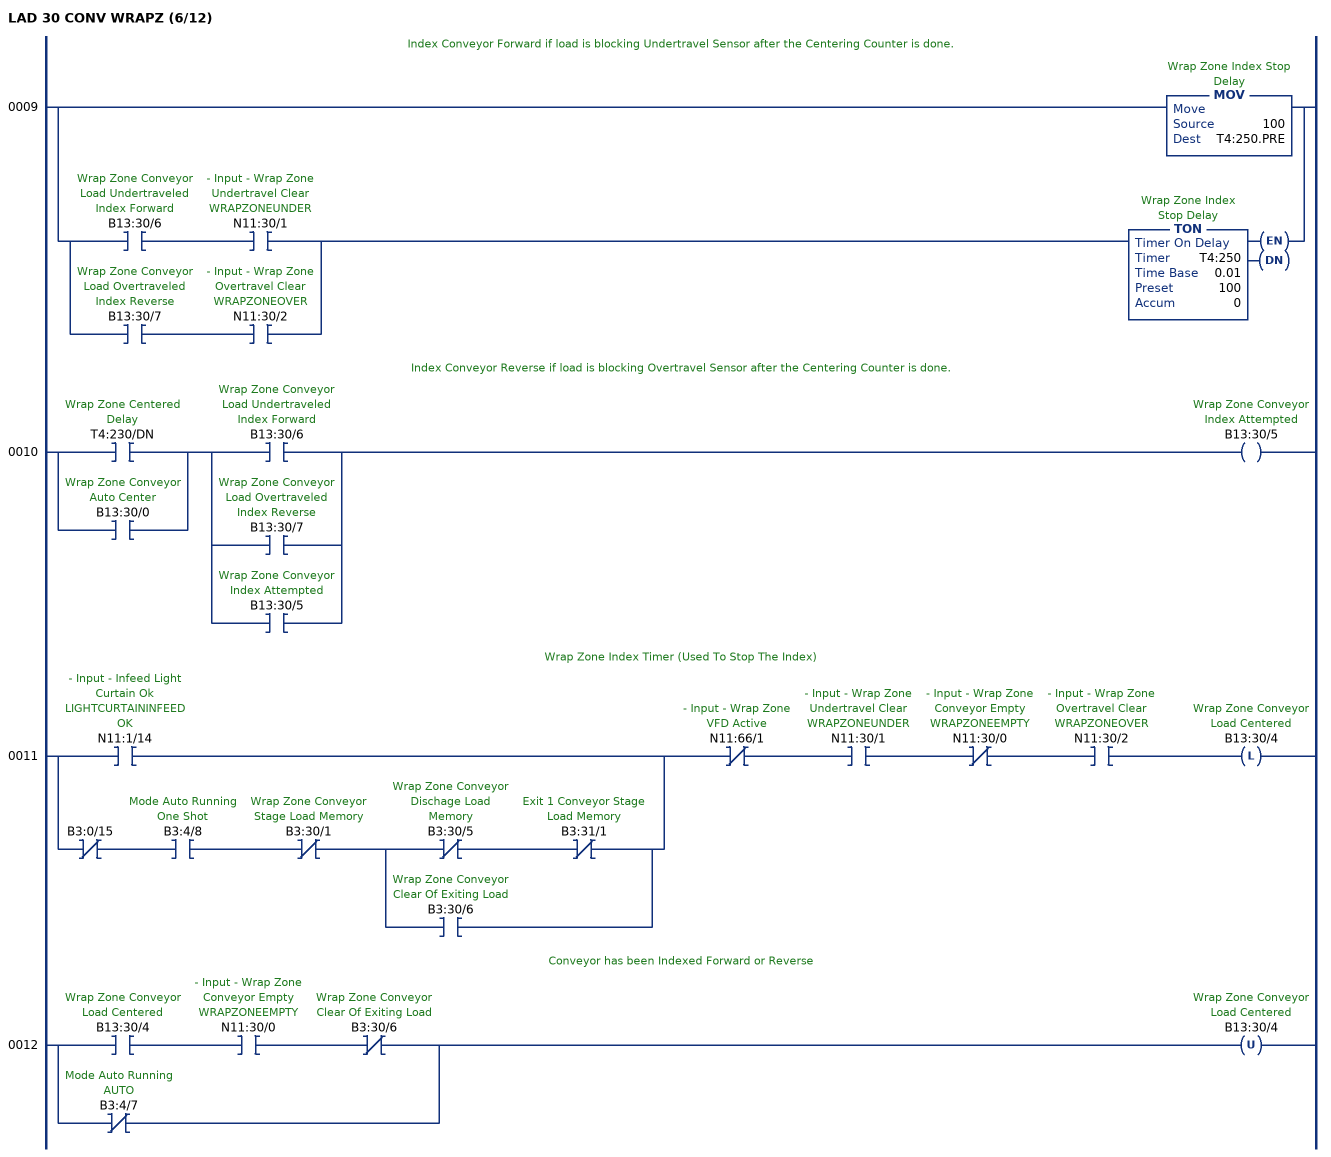
% Rung: 9 %
% Index Conveyor Forward if load is blocking Undertravel Sensor after the Centering Counter is done. %
SOR BST MOV 100 T4:250.PRE NXB BST XIC B13:30/6 XIC N11:30/1 NXB XIC B13:30/7 XIC N11:30/2 BND TON T4:250 0.01 100 0 BND EOR
%   T4:250  "Wrap Zone Index Stop Delay" %
%   B13:30/6  "Wrap Zone Conveyor Load Undertraveled Index Forward" %
%   N11:30/1  WRAPZONEUNDER  "- Input - Wrap Zone Undertravel Clear" %
%   B13:30/7  "Wrap Zone Conveyor Load Overtraveled Index Reverse" %
%   N11:30/2  WRAPZONEOVER  "- Input - Wrap Zone Overtravel Clear" %
% Rung: 10 %
% Index Conveyor Reverse if load is blocking Overtravel Sensor after the Centering Counter is done. %
SOR BST XIC T4:230/DN NXB XIC B13:30/0 BND BST XIC B13:30/6 NXB XIC B13:30/7 NXB XIC B13:30/5 BND OTE B13:30/5 EOR
%   T4:230  "Wrap Zone Centered Delay" %
%   B13:30/0  "Wrap Zone Conveyor Auto Center" %
%   B13:30/6  "Wrap Zone Conveyor Load Undertraveled Index Forward" %
%   B13:30/7  "Wrap Zone Conveyor Load Overtraveled Index Reverse" %
%   B13:30/5  "Wrap Zone Conveyor Index Attempted" %
% Rung: 11 %
% Wrap Zone Index Timer (Used To Stop The Index) %
SOR BST XIC N11:1/14 NXB XIO B3:0/15 XIC B3:4/8 XIO B3:30/1 BST XIO B3:30/5 XIO B3:31/1 NXB XIC B3:30/6 BND BND XIO N11:66/1 XIC N11:30/1 XIO N11:30/0 XIC N11:30/2 OTL B13:30/4 EOR
%   N11:1/14  LIGHTCURTAININFEEDOK  "- Input - Infeed Light Curtain Ok" %
%   B3:4/8  "Mode Auto Running One Shot" %
%   B3:30/1  "Wrap Zone Conveyor Stage Load Memory" %
%   B3:30/5  "Wrap Zone Conveyor Dischage Load Memory" %
%   B3:31/1  "Exit 1 Conveyor Stage Load Memory" %
%   B3:30/6  "Wrap Zone Conveyor Clear Of Exiting Load" %
%   N11:66/1  "- Input - Wrap Zone VFD Active" %
%   N11:30/1  WRAPZONEUNDER  "- Input - Wrap Zone Undertravel Clear" %
%   N11:30/0  WRAPZONEEMPTY  "- Input - Wrap Zone Conveyor Empty" %
%   N11:30/2  WRAPZONEOVER  "- Input - Wrap Zone Overtravel Clear" %
%   B13:30/4  "Wrap Zone Conveyor Load Centered" %
% Rung: 12 %
% Conveyor has been Indexed Forward or Reverse %
SOR BST XIC B13:30/4 XIC N11:30/0 XIO B3:30/6 NXB XIO B3:4/7 BND OTU B13:30/4 EOR
%   B13:30/4  "Wrap Zone Conveyor Load Centered" %
%   N11:30/0  WRAPZONEEMPTY  "- Input - Wrap Zone Conveyor Empty" %
%   B3:30/6  "Wrap Zone Conveyor Clear Of Exiting Load" %
%   B3:4/7  AUTO  "Mode Auto Running" %

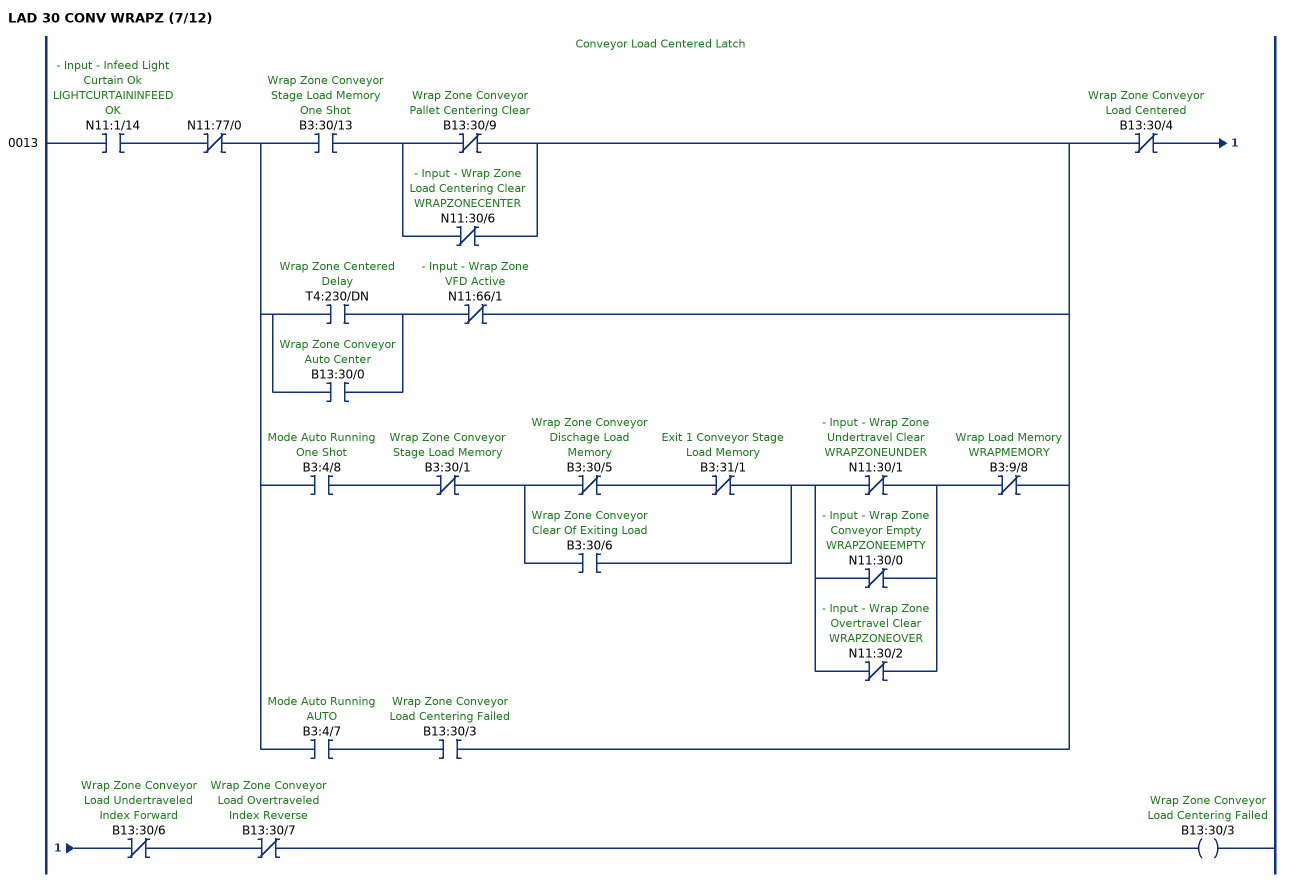
% Rung: 13 %
% Conveyor Load Centered Latch %
SOR XIC N11:1/14 XIO N11:77/0 BST XIC B3:30/13 BST XIO B13:30/9 NXB XIO N11:30/6 BND NXB BST XIC T4:230/DN NXB XIC B13:30/0 BND XIO N11:66/1 NXB XIC B3:4/8 XIO B3:30/1 BST XIO B3:30/5 XIO B3:31/1 NXB XIC B3:30/6 BND BST XIO N11:30/1 NXB XIO N11:30/0 NXB XIO N11:30/2 BND XIO B3:9/8 NXB XIC B3:4/7 XIC B13:30/3 BND XIO B13:30/4 XIO B13:30/6 XIO B13:30/7 OTE B13:30/3 EOR
%   N11:1/14  LIGHTCURTAININFEEDOK  "- Input - Infeed Light Curtain Ok" %
%   B3:30/13  "Wrap Zone Conveyor Stage Load Memory One Shot" %
%   B13:30/9  "Wrap Zone Conveyor Pallet Centering Clear" %
%   N11:30/6  WRAPZONECENTER  "- Input - Wrap Zone Load Centering Clear" %
%   T4:230  "Wrap Zone Centered Delay" %
%   B13:30/0  "Wrap Zone Conveyor Auto Center" %
%   N11:66/1  "- Input - Wrap Zone VFD Active" %
%   B3:4/8  "Mode Auto Running One Shot" %
%   B3:30/1  "Wrap Zone Conveyor Stage Load Memory" %
%   B3:30/5  "Wrap Zone Conveyor Dischage Load Memory" %
%   B3:31/1  "Exit 1 Conveyor Stage Load Memory" %
%   B3:30/6  "Wrap Zone Conveyor Clear Of Exiting Load" %
%   N11:30/1  WRAPZONEUNDER  "- Input - Wrap Zone Undertravel Clear" %
%   N11:30/0  WRAPZONEEMPTY  "- Input - Wrap Zone Conveyor Empty" %
%   N11:30/2  WRAPZONEOVER  "- Input - Wrap Zone Overtravel Clear" %
%   B3:9/8  WRAPMEMORY  "Wrap Load Memory" %
%   B3:4/7  AUTO  "Mode Auto Running" %
%   B13:30/3  "Wrap Zone Conveyor Load Centering Failed" %
%   B13:30/4  "Wrap Zone Conveyor Load Centered" %
%   B13:30/6  "Wrap Zone Conveyor Load Undertraveled Index Forward" %
%   B13:30/7  "Wrap Zone Conveyor Load Overtraveled Index Reverse" %

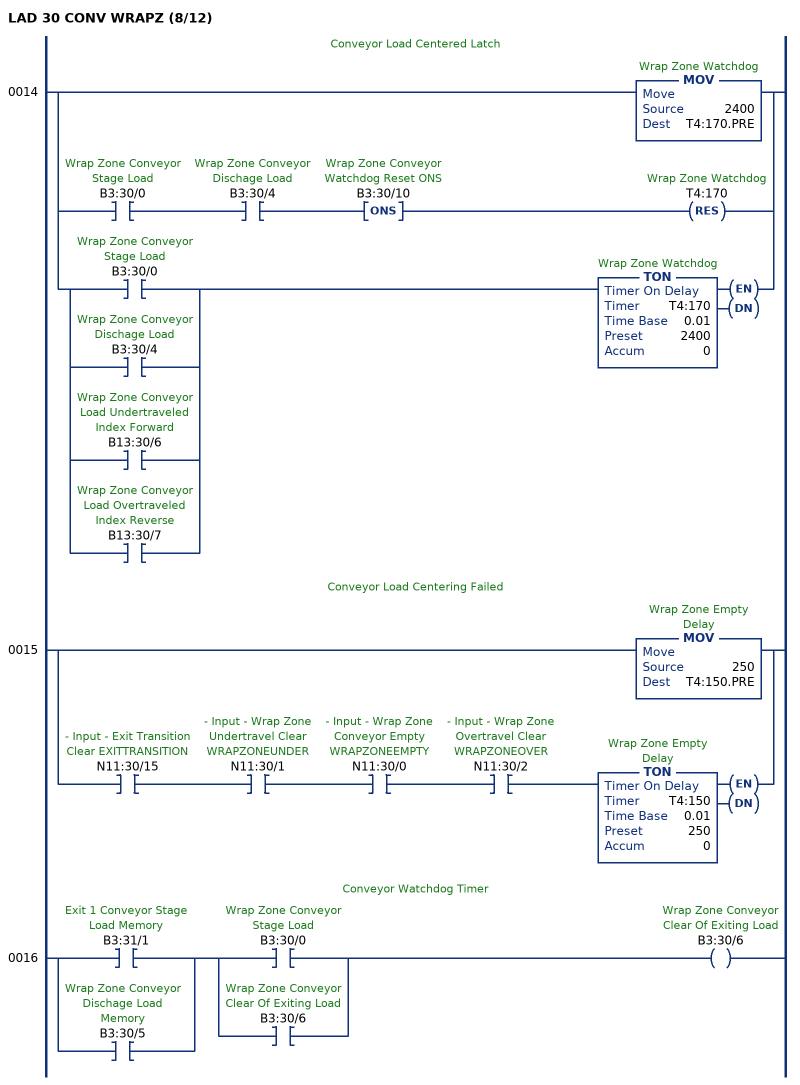
% Rung: 14 %
% Conveyor Load Centered Latch %
SOR BST MOV 2400 T4:170.PRE NXB XIC B3:30/0 XIC B3:30/4 ONS B3:30/10 RES T4:170 NXB BST XIC B3:30/0 NXB XIC B3:30/4 NXB XIC B13:30/6 NXB XIC B13:30/7 BND TON T4:170 0.01 2400 0 BND EOR
%   T4:170  "Wrap Zone Watchdog" %
%   B3:30/0  "Wrap Zone Conveyor Stage Load" %
%   B3:30/4  "Wrap Zone Conveyor Dischage Load" %
%   B3:30/10  "Wrap Zone Conveyor Watchdog Reset ONS" %
%   B13:30/6  "Wrap Zone Conveyor Load Undertraveled Index Forward" %
%   B13:30/7  "Wrap Zone Conveyor Load Overtraveled Index Reverse" %
% Rung: 15 %
% Conveyor Load Centering Failed %
SOR BST MOV 250 T4:150.PRE NXB XIC N11:30/15 XIC N11:30/1 XIC N11:30/0 XIC N11:30/2 TON T4:150 0.01 250 0 BND EOR
%   T4:150  "Wrap Zone Empty Delay" %
%   N11:30/15  EXITTRANSITION  "- Input - Exit Transition Clear" %
%   N11:30/1  WRAPZONEUNDER  "- Input - Wrap Zone Undertravel Clear" %
%   N11:30/0  WRAPZONEEMPTY  "- Input - Wrap Zone Conveyor Empty" %
%   N11:30/2  WRAPZONEOVER  "- Input - Wrap Zone Overtravel Clear" %
% Rung: 16 %
% Conveyor Watchdog Timer %
SOR BST XIC B3:31/1 NXB XIC B3:30/5 BND BST XIC B3:30/0 NXB XIC B3:30/6 BND OTE B3:30/6 EOR
%   B3:31/1  "Exit 1 Conveyor Stage Load Memory" %
%   B3:30/5  "Wrap Zone Conveyor Dischage Load Memory" %
%   B3:30/0  "Wrap Zone Conveyor Stage Load" %
%   B3:30/6  "Wrap Zone Conveyor Clear Of Exiting Load" %

